LIN {X 0,Y 411.148,Z 377.722,A -85,B 0,C 180,E1 -10646.387,E2 -10646.387} C_VEL
LIN {X 0,Y 411.477,Z 371.571,A -85,B 0,C 180,E1 -10649.691,E2 -10649.691} C_VEL
LIN {X 0,Y 411.355,Z 369.248,A -85,B 0,C 180,E1 -10651.013,E2 -10651.013} C_VEL
LIN {X 0,Y 411.215,Z 369.265,A -85,B 0,C 180,E1 -10654.879,E2 -10654.879} C_VEL
LIN {X 0,Y 411.214,Z 369.262,A -85,B 0,C 180,E1 -10658.17,E2 -10658.17} C_VEL
LIN {X 0,Y 411.167,Z 369.269,A -85,B 0,C 180,E1 -10661.228,E2 -10661.228} C_VEL
LIN {X 0,Y 411.18,Z 369.267,A -85,B 0,C 180,E1 -10664.49,E2 -10664.49} C_VEL
LIN {X 0,Y 411.182,Z 369.267,A -85,B 0,C 180,E1 -10668.195,E2 -10668.195} C_VEL
LIN {X 0,Y 411.22,Z 369.263,A -85,B 0,C 180,E1 -10670.776,E2 -10670.776} C_VEL
LIN {X 0,Y 411.201,Z 369.266,A -85,B 0,C 180,E1 -10674.471,E2 -10674.471} C_VEL
LIN {X 0,Y 411.21,Z 369.263,A -85,B 0,C 180,E1 -10676.873,E2 -10676.873} C_VEL
LIN {X 0,Y 411.236,Z 369.261,A -85,B 0,C 180,E1 -10680.644,E2 -10680.644} C_VEL
LIN {X 0,Y 411.24,Z 369.258,A -85,B 0,C 180,E1 -10683.619,E2 -10683.619} C_VEL
LIN {X 0,Y 411.206,Z 369.263,A -85,B 0,C 180,E1 -10686.852,E2 -10686.852} C_VEL
LIN {X 0,Y 411.219,Z 369.264,A -85,B 0,C 180,E1 -10690.05,E2 -10690.05} C_VEL
LIN {X 0,Y 411.267,Z 369.255,A -85,B 0,C 180,E1 -10693.131,E2 -10693.131} C_VEL
LIN {X 0,Y 411.309,Z 369.248,A -85,B 0,C 180,E1 -10696.896,E2 -10696.896} C_VEL
LIN {X 0,Y 411.296,Z 369.254,A -85,B 0,C 180,E1 -10700.161,E2 -10700.161} C_VEL
LIN {X 0,Y 411.456,Z 369.232,A -85,B 0,C 180,E1 -10703.133,E2 -10703.133} C_VEL
LIN {X 0,Y 411.313,Z 369.249,A -85,B 0,C 180,E1 -10705.099,E2 -10705.099} C_VEL
LIN {X 0,Y 411.515,Z 369.228,A -85,B 0,C 180,E1 -10708.042,E2 -10708.042} C_VEL
LIN {X 0,Y 411.644,Z 369.211,A -85,B 0,C 180,E1 -10710,E2 -10710} C_VEL
LIN {X 0,Y 411.469,Z 369.23,A -85,B 0,C 180,E1 -10712.937,E2 -10712.937} C_VEL
LIN {X 0,Y 411.455,Z 369.231,A -85,B 0,C 180,E1 -10716.867,E2 -10716.867} C_VEL
LIN {X 0,Y 411.308,Z 369.253,A -85,B 0,C 180,E1 -10719.838,E2 -10719.838} C_VEL
LIN {X 0,Y 411.309,Z 369.25,A -85,B 0,C 180,E1 -10723.104,E2 -10723.104} C_VEL
LIN {X 0,Y 411.259,Z 369.255,A -85,B 0,C 180,E1 -10726.756,E2 -10726.756} C_VEL
LIN {X 0,Y 410.624,Z 369.339,A -85,B 0,C 180,E1 -10727.574,E2 -10727.574} C_VEL
LIN {X 0,Y 407.754,Z 369.691,A -85,B 0,C 180,E1 -10728.902,E2 -10728.902} C_VEL
LIN {X 0,Y 405.301,Z 369.999,A -85,B 0,C 180,E1 -10729.974,E2 -10729.974} C_VEL
LIN {X 0,Y 404.247,Z 370.128,A -85,B 0,C 180,E1 -10730.804,E2 -10730.804} C_VEL
LIN {X 0,Y 404.162,Z 370.14,A -85,B 0,C 180,E1 -10731.085,E2 -10731.085} C_VEL
LIN {X 0,Y 404.18,Z 370.138,A -85,B 0,C 180,E1 -10734.665,E2 -10734.665} C_VEL
LIN {X 0,Y 404.198,Z 370.137,A -85,B 0,C 180,E1 -10737.999,E2 -10737.999} C_VEL
LIN {X 0,Y 404.142,Z 370.145,A -85,B 0,C 180,E1 -10741.558,E2 -10741.558} C_VEL
LIN {X 0,Y 404.187,Z 370.139,A -85,B 0,C 180,E1 -10745.016,E2 -10745.016} C_VEL
LIN {X 0,Y 404.16,Z 370.141,A -85,B 0,C 180,E1 -10748.756,E2 -10748.756} C_VEL
LIN {X 0,Y 404.126,Z 370.146,A -85,B 0,C 180,E1 -10751.6,E2 -10751.6} C_VEL
LIN {X 0,Y 404.148,Z 370.142,A -85,B 0,C 180,E1 -10754.522,E2 -10754.522} C_VEL
LIN {X 0,Y 404.139,Z 370.145,A -85,B 0,C 180,E1 -10757.296,E2 -10757.296} C_VEL
LIN {X 0,Y 404.171,Z 370.139,A -85,B 0,C 180,E1 -10759.955,E2 -10759.955} C_VEL
LIN {X 0,Y 404.139,Z 370.147,A -85,B 0,C 180,E1 -10763.125,E2 -10763.125} C_VEL
LIN {X 0,Y 404.147,Z 370.142,A -85,B 0,C 180,E1 -10766.188,E2 -10766.188} C_VEL
LIN {X 0,Y 404.148,Z 370.142,A -85,B 0,C 180,E1 -10769.715,E2 -10769.715} C_VEL
LIN {X 0,Y 404.198,Z 370.138,A -85,B 0,C 180,E1 -10773.123,E2 -10773.123} C_VEL
LIN {X 0,Y 404.18,Z 370.138,A -85,B 0,C 180,E1 -10775.334,E2 -10775.334} C_VEL
LIN {X 0,Y 404.142,Z 370.145,A -85,B 0,C 180,E1 -10778.581,E2 -10778.581} C_VEL
LIN {X 0,Y 404.213,Z 370.133,A -85,B 0,C 180,E1 -10781.762,E2 -10781.762} C_VEL
LIN {X 0,Y 404.21,Z 370.137,A -85,B 0,C 180,E1 -10784.882,E2 -10784.882} C_VEL
LIN {X 0,Y 404.273,Z 370.126,A -85,B 0,C 180,E1 -10787.959,E2 -10787.959} C_VEL
LIN {X 0,Y 404.436,Z 370.107,A -85,B 0,C 180,E1 -10792.1,E2 -10792.1} C_VEL
LIN {X 0,Y 404.426,Z 370.107,A -85,B 0,C 180,E1 -10794.015,E2 -10794.015} C_VEL
LIN {X 0,Y 404.483,Z 370.101,A -85,B 0,C 180,E1 -10798.008,E2 -10798.008} C_VEL
LIN {X 0,Y 404.614,Z 370.085,A -85,B 0,C 180,E1 -10800,E2 -10800} C_VEL
LIN {X 0,Y 404.425,Z 370.108,A -85,B 0,C 180,E1 -10802.988,E2 -10802.988} C_VEL
LIN {X 0,Y 404.414,Z 370.108,A -85,B 0,C 180,E1 -10806.987,E2 -10806.987} C_VEL
LIN {X 0,Y 404.261,Z 370.13,A -85,B 0,C 180,E1 -10810.012,E2 -10810.012} C_VEL
LIN {X 0,Y 404.268,Z 370.127,A -85,B 0,C 180,E1 -10813.211,E2 -10813.211} C_VEL
LIN {X 0,Y 404.218,Z 370.132,A -85,B 0,C 180,E1 -10817.007,E2 -10817.007} C_VEL
LIN {X 0,Y 404.166,Z 370.141,A -85,B 0,C 180,E1 -10820.351,E2 -10820.351} C_VEL
LIN {X 0,Y 404.171,Z 370.14,A -85,B 0,C 180,E1 -10823.574,E2 -10823.574} C_VEL
LIN {X 0,Y 404.185,Z 370.138,A -85,B 0,C 180,E1 -10825.766,E2 -10825.766} C_VEL
LIN {X 0,Y 404.197,Z 370.139,A -85,B 0,C 180,E1 -10828,E2 -10828} C_VEL
LIN {X 0,Y 404.141,Z 370.144,A -85,B 0,C 180,E1 -10831.558,E2 -10831.558} C_VEL
LIN {X 0,Y 404.187,Z 370.137,A -85,B 0,C 180,E1 -10835.016,E2 -10835.016} C_VEL
LIN {X 0,Y 404.161,Z 370.139,A -85,B 0,C 180,E1 -10838.756,E2 -10838.756} C_VEL
LIN {X 0,Y 404.143,Z 370.145,A -85,B 0,C 180,E1 -10841.603,E2 -10841.603} C_VEL
LIN {X 0,Y 404.152,Z 370.142,A -85,B 0,C 180,E1 -10844.523,E2 -10844.523} C_VEL
LIN {X 0,Y 404.141,Z 370.144,A -85,B 0,C 180,E1 -10847.296,E2 -10847.296} C_VEL
LIN {X 0,Y 404.17,Z 370.14,A -85,B 0,C 180,E1 -10849.955,E2 -10849.955} C_VEL
LIN {X 0,Y 404.18,Z 370.14,A -85,B 0,C 180,E1 -10853.758,E2 -10853.758} C_VEL
LIN {X 0,Y 404.188,Z 370.32,A -85,B 0,C 180,E1 -10854.162,E2 -10854.162} C_VEL
LIN {X 0,Y 406.436,Z 380.828,A -85,B 0,C 180,E1 -10857.291,E2 -10857.291} C_VEL
LIN {X 0,Y 408.438,Z 390.536,A -85,B 0,C 180,E1 -10860.066,E2 -10860.066} C_VEL
LIN {X 0,Y 408.583,Z 393.722,A -85,B 0,C 180,E1 -10860.927,E2 -10860.927} C_VEL
LIN {X 0,Y 407.037,Z 407.44,A -85,B 0,C 180,E1 -10864.427,E2 -10864.427} C_VEL
LIN {X 0,Y 405.68,Z 422.214,A -85,B 0,C 180,E1 -10868.132,E2 -10868.132} C_VEL
LIN {X 0,Y 404.511,Z 439.114,A -85,B 0,C 180,E1 -10872.299,E2 -10872.299} C_VEL
LIN {X 0,Y 404.238,Z 443.217,A -85,B 0,C 180,E1 -10873.301,E2 -10873.301} C_VEL
LIN {X 0,Y 405.63,Z 458.581,A -85,B 0,C 180,E1 -10873.82,E2 -10873.82} C_VEL
LIN {X 0,Y 406.354,Z 470.143,A -85,B 0,C 180,E1 -10874.386,E2 -10874.386} C_VEL
LIN {X 0,Y 405.709,Z 482.837,A -85,B 0,C 180,E1 -10875.196,E2 -10875.196} C_VEL
LIN {X 0,Y 405.185,Z 494.035,A -85,B 0,C 180,E1 -10876.131,E2 -10876.131} C_VEL
LIN {X 0,Y 404.711,Z 503.184,A -85,B 0,C 180,E1 -10877.081,E2 -10877.081} C_VEL
LIN {X 0,Y 404.142,Z 512.126,A -85,B 0,C 180,E1 -10878.21,E2 -10878.21} C_VEL
LIN {X 0,Y 403.682,Z 520.303,A -85,B 0,C 180,E1 -10879.467,E2 -10879.467} C_VEL
LIN {X 0,Y 403.357,Z 528.26,A -85,B 0,C 180,E1 -10880.978,E2 -10880.978} C_VEL
LIN {X 0,Y 403.201,Z 534.531,A -85,B 0,C 180,E1 -10882.488,E2 -10882.488} C_VEL
LIN {X 0,Y 403.139,Z 539.444,A -85,B 0,C 180,E1 -10883.996,E2 -10883.996} C_VEL
LIN {X 0,Y 403.099,Z 543.144,A -85,B 0,C 180,E1 -10885.5,E2 -10885.5} C_VEL
LIN {X 0,Y 403.268,Z 545.764,A -85,B 0,C 180,E1 -10887.003,E2 -10887.003} C_VEL
LIN {X 0,Y 403.223,Z 546.939,A -85,B 0,C 180,E1 -10888.002,E2 -10888.002} C_VEL
LIN {X 0,Y 403.121,Z 547.631,A -85,B 0,C 180,E1 -10889.001,E2 -10889.001} C_VEL
LIN {X 0,Y 403.102,Z 547.906,A -85,B 0,C 180,E1 -10890,E2 -10890} C_VEL
LIN {X 0,Y 403.123,Z 547.774,A -85,B 0,C 180,E1 -10890.999,E2 -10890.999} C_VEL
LIN {X 0,Y 403.218,Z 547.196,A -85,B 0,C 180,E1 -10891.998,E2 -10891.998} C_VEL
LIN {X 0,Y 403.204,Z 546.167,A -85,B 0,C 180,E1 -10892.998,E2 -10892.998} C_VEL
LIN {X 0,Y 403.116,Z 544.713,A -85,B 0,C 180,E1 -10893.999,E2 -10893.999} C_VEL
LIN {X 0,Y 403.111,Z 541.666,A -85,B 0,C 180,E1 -10895.503,E2 -10895.503} C_VEL
LIN {X 0,Y 403.183,Z 537.532,A -85,B 0,C 180,E1 -10897.009,E2 -10897.009} C_VEL
LIN {X 0,Y 403.332,Z 531.141,A -85,B 0,C 180,E1 -10898.77,E2 -10898.77} C_VEL
LIN {X 0,Y 403.59,Z 524.167,A -85,B 0,C 180,E1 -10900.282,E2 -10900.282} C_VEL
LIN {X 0,Y 404.107,Z 517.08,A -85,B 0,C 180,E1 -10901.537,E2 -10901.537} C_VEL
LIN {X 0,Y 404.66,Z 508.52,A -85,B 0,C 180,E1 -10902.794,E2 -10902.794} C_VEL
LIN {X 0,Y 405.427,Z 497.96,A -85,B 0,C 180,E1 -10904.045,E2 -10904.045} C_VEL
LIN {X 0,Y 406.179,Z 487.574,A -85,B 0,C 180,E1 -10905.043,E2 -10905.043} C_VEL
LIN {X 0,Y 406.997,Z 476.089,A -85,B 0,C 180,E1 -10905.91,E2 -10905.91} C_VEL
LIN {X 0,Y 407.201,Z 467.052,A -85,B 0,C 180,E1 -10906.469,E2 -10906.469} C_VEL
LIN {X 0,Y 406.365,Z 453.454,A -85,B 0,C 180,E1 -10907.152,E2 -10907.152} C_VEL
LIN {X 0,Y 404.671,Z 441.819,A -85,B 0,C 180,E1 -10907.628,E2 -10907.628} C_VEL
LIN {X 0,Y 405.657,Z 428.844,A -85,B 0,C 180,E1 -10910.914,E2 -10910.914} C_VEL
LIN {X 0,Y 406.916,Z 417.346,A -85,B 0,C 180,E1 -10914,E2 -10914} C_VEL
LIN {X 0,Y 408.565,Z 406.517,A -85,B 0,C 180,E1 -10917.119,E2 -10917.119} C_VEL
LIN {X 0,Y 409.97,Z 399.423,A -85,B 0,C 180,E1 -10919.308,E2 -10919.308} C_VEL
LIN {X 0,Y 410.147,Z 396.422,A -85,B 0,C 180,E1 -10920.364,E2 -10920.364} C_VEL
LIN {X 0,Y 408.861,Z 389.269,A -85,B 0,C 180,E1 -10923.371,E2 -10923.371} C_VEL
LIN {X 0,Y 407.709,Z 384.465,A -85,B 0,C 180,E1 -10925.887,E2 -10925.887} C_VEL
LIN {X 0,Y 406.605,Z 379.983,A -85,B 0,C 180,E1 -10928.94,E2 -10928.94} C_VEL
LIN {X 0,Y 406.056,Z 377.657,A -85,B 0,C 180,E1 -10931.125,E2 -10931.125} C_VEL
LIN {X 0,Y 405.542,Z 375.828,A -85,B 0,C 180,E1 -10933.884,E2 -10933.884} C_VEL
LIN {X 0,Y 405.371,Z 375.113,A -85,B 0,C 180,E1 -10936.733,E2 -10936.733} C_VEL
LIN {X 0,Y 405.424,Z 375.549,A -85,B 0,C 180,E1 -10939.707,E2 -10939.707} C_VEL
LIN {X 0,Y 405.674,Z 377.131,A -85,B 0,C 180,E1 -10942.837,E2 -10942.837} C_VEL
LIN {X 0,Y 406.006,Z 378.918,A -85,B 0,C 180,E1 -10945.164,E2 -10945.164} C_VEL
LIN {X 0,Y 406.357,Z 381.647,A -85,B 0,C 180,E1 -10947.937,E2 -10947.937} C_VEL
LIN {X 0,Y 406.342,Z 383.966,A -85,B 0,C 180,E1 -10949.896,E2 -10949.896} C_VEL
LIN {X 0,Y 405.779,Z 388.489,A -85,B 0,C 180,E1 -10953.236,E2 -10953.236} C_VEL
LIN {X 0,Y 405.249,Z 393.854,A -85,B 0,C 180,E1 -10956.803,E2 -10956.803} C_VEL
LIN {X 0,Y 404.742,Z 400.152,A -85,B 0,C 180,E1 -10960.736,E2 -10960.736} C_VEL
LIN {X 0,Y 404.373,Z 405.404,A -85,B 0,C 180,E1 -10963.854,E2 -10963.854} C_VEL
LIN {X 0,Y 404.048,Z 412.145,A -85,B 0,C 180,E1 -10967.697,E2 -10967.697} C_VEL
LIN {X 0,Y 404.018,Z 412.616,A -85,B 0,C 180,E1 -10967.951,E2 -10967.951} C_VEL
LIN {X 0,Y 406.519,Z 423.605,A -85,B 0,C 180,E1 -10968.785,E2 -10968.785} C_VEL
LIN {X 0,Y 407.207,Z 428.2,A -85,B 0,C 180,E1 -10969.182,E2 -10969.182} C_VEL
LIN {X 0,Y 406.611,Z 437.638,A -85,B 0,C 180,E1 -10970.047,E2 -10970.047} C_VEL
LIN {X 0,Y 405.969,Z 446.024,A -85,B 0,C 180,E1 -10971.037,E2 -10971.037} C_VEL
LIN {X 0,Y 405.274,Z 454.119,A -85,B 0,C 180,E1 -10972.276,E2 -10972.276} C_VEL
LIN {X 0,Y 404.79,Z 460.311,A -85,B 0,C 180,E1 -10973.52,E2 -10973.52} C_VEL
LIN {X 0,Y 404.377,Z 464.194,A -85,B 0,C 180,E1 -10974.515,E2 -10974.515} C_VEL
LIN {X 0,Y 404.143,Z 467.219,A -85,B 0,C 180,E1 -10975.512,E2 -10975.512} C_VEL
LIN {X 0,Y 403.552,Z 470.386,A -85,B 0,C 180,E1 -10977.005,E2 -10977.005} C_VEL
LIN {X 0,Y 403.365,Z 471.602,A -85,B 0,C 180,E1 -10978.003,E2 -10978.003} C_VEL
LIN {X 0,Y 403.255,Z 472.146,A -85,B 0,C 180,E1 -10979.001,E2 -10979.001} C_VEL
LIN {X 0,Y 403.193,Z 472.025,A -85,B 0,C 180,E1 -10980,E2 -10980} C_VEL
LIN {X 0,Y 403.192,Z 471.236,A -85,B 0,C 180,E1 -10980.999,E2 -10980.999} C_VEL
LIN {X 0,Y 403.346,Z 468.774,A -85,B 0,C 180,E1 -10982.497,E2 -10982.497} C_VEL
LIN {X 0,Y 403.608,Z 466.231,A -85,B 0,C 180,E1 -10983.494,E2 -10983.494} C_VEL
LIN {X 0,Y 403.853,Z 460.925,A -85,B 0,C 180,E1 -10984.992,E2 -10984.992} C_VEL
LIN {X 0,Y 404.041,Z 454.874,A -85,B 0,C 180,E1 -10986.241,E2 -10986.241} C_VEL
LIN {X 0,Y 404.249,Z 447.598,A -85,B 0,C 180,E1 -10987.399,E2 -10987.399} C_VEL
LIN {X 0,Y 404.594,Z 438.691,A -85,B 0,C 180,E1 -10988.491,E2 -10988.491} C_VEL
LIN {X 0,Y 404.977,Z 429.418,A -85,B 0,C 180,E1 -10989.363,E2 -10989.363} C_VEL
LIN {X 0,Y 405.109,Z 422.751,A -85,B 0,C 180,E1 -10989.864,E2 -10989.864} C_VEL
LIN {X 0,Y 403.584,Z 411.764,A -85,B 0,C 180,E1 -10990.536,E2 -10990.536} C_VEL
LIN {X 0,Y 403.201,Z 408.969,A -85,B 0,C 180,E1 -10990.673,E2 -10990.673} C_VEL
LIN {X 0,Y 403.341,Z 403.119,A -85,B 0,C 180,E1 -10993.605,E2 -10993.605} C_VEL
LIN {X 0,Y 403.527,Z 397.076,A -85,B 0,C 180,E1 -10996.683,E2 -10996.683} C_VEL
LIN {X 0,Y 403.733,Z 389.969,A -85,B 0,C 180,E1 -11000.374,E2 -11000.374} C_VEL
LIN {X 0,Y 403.888,Z 383.868,A -85,B 0,C 180,E1 -11003.592,E2 -11003.592} C_VEL
LIN {X 0,Y 404.111,Z 377.71,A -85,B 0,C 180,E1 -11006.883,E2 -11006.883} C_VEL
LIN {X 0,Y 404.505,Z 371.515,A -85,B 0,C 180,E1 -11010.256,E2 -11010.256} C_VEL
LIN {X 0,Y 404.318,Z 370.125,A -85,B 0,C 180,E1 -11011.14,E2 -11011.14} C_VEL
LIN {X 0,Y 404.185,Z 370.138,A -85,B 0,C 180,E1 -11015.19,E2 -11015.19} C_VEL
LIN {X 0,Y 404.161,Z 370.142,A -85,B 0,C 180,E1 -11018.756,E2 -11018.756} C_VEL
LIN {X 0,Y 404.126,Z 370.144,A -85,B 0,C 180,E1 -11021.6,E2 -11021.6} C_VEL
LIN {X 0,Y 404.15,Z 370.144,A -85,B 0,C 180,E1 -11024.522,E2 -11024.522} C_VEL
LIN {X 0,Y 404.143,Z 370.143,A -85,B 0,C 180,E1 -11027.296,E2 -11027.296} C_VEL
LIN {X 0,Y 404.172,Z 370.139,A -85,B 0,C 180,E1 -11029.955,E2 -11029.955} C_VEL
LIN {X 0,Y 404.139,Z 370.143,A -85,B 0,C 180,E1 -11033.125,E2 -11033.125} C_VEL
LIN {X 0,Y 404.148,Z 370.143,A -85,B 0,C 180,E1 -11036.188,E2 -11036.188} C_VEL
LIN {X 0,Y 404.149,Z 370.142,A -85,B 0,C 180,E1 -11039.715,E2 -11039.715} C_VEL
LIN {X 0,Y 404.198,Z 370.135,A -85,B 0,C 180,E1 -11043.123,E2 -11043.123} C_VEL
LIN {X 0,Y 404.18,Z 370.136,A -85,B 0,C 180,E1 -11045.334,E2 -11045.334} C_VEL
LIN {X 0,Y 404.142,Z 370.144,A -85,B 0,C 180,E1 -11048.581,E2 -11048.581} C_VEL
LIN {X 0,Y 404.214,Z 370.135,A -85,B 0,C 180,E1 -11051.762,E2 -11051.762} C_VEL
LIN {X 0,Y 404.21,Z 370.134,A -85,B 0,C 180,E1 -11054.882,E2 -11054.882} C_VEL
LIN {X 0,Y 404.26,Z 370.13,A -85,B 0,C 180,E1 -11057.958,E2 -11057.958} C_VEL
LIN {X 0,Y 404.408,Z 370.111,A -85,B 0,C 180,E1 -11062.129,E2 -11062.129} C_VEL
LIN {X 0,Y 404.423,Z 370.109,A -85,B 0,C 180,E1 -11064.015,E2 -11064.015} C_VEL
LIN {X 0,Y 404.484,Z 370.104,A -85,B 0,C 180,E1 -11068.008,E2 -11068.008} C_VEL
LIN {X 0,Y 404.613,Z 370.087,A -85,B 0,C 180,E1 -11070,E2 -11070} C_VEL
LIN {X 0,Y 404.426,Z 370.107,A -85,B 0,C 180,E1 -11072.988,E2 -11072.988} C_VEL
LIN {X 0,Y 404.403,Z 370.109,A -85,B 0,C 180,E1 -11076.987,E2 -11076.987} C_VEL
LIN {X 0,Y 404.27,Z 370.128,A -85,B 0,C 180,E1 -11080.011,E2 -11080.011} C_VEL
LIN {X 0,Y 404.27,Z 370.128,A -85,B 0,C 180,E1 -11083.211,E2 -11083.211} C_VEL
LIN {X 0,Y 404.219,Z 370.133,A -85,B 0,C 180,E1 -11087.007,E2 -11087.007} C_VEL
LIN {X 0,Y 404.201,Z 370.134,A -85,B 0,C 180,E1 -11090.35,E2 -11090.35} C_VEL
LIN {X 0,Y 404.162,Z 370.14,A -85,B 0,C 180,E1 -11091.085,E2 -11091.085} C_VEL
LIN {X 0,Y 403.499,Z 370.226,A -85,B 0,C 180,E1 -11091.917,E2 -11091.917} C_VEL
LIN {X 0,Y 400.656,Z 370.581,A -85,B 0,C 180,E1 -11093.27,E2 -11093.27} C_VEL
LIN {X 0,Y 398.255,Z 370.877,A -85,B 0,C 180,E1 -11094.362,E2 -11094.362} C_VEL
LIN {X 0,Y 397.234,Z 371.006,A -85,B 0,C 180,E1 -11095.207,E2 -11095.207} C_VEL
LIN {X 0,Y 397.156,Z 371.015,A -85,B 0,C 180,E1 -11095.493,E2 -11095.493} C_VEL
LIN {X 0,Y 397.125,Z 371.016,A -85,B 0,C 180,E1 -11098.543,E2 -11098.543} C_VEL
LIN {X 0,Y 397.081,Z 371.022,A -85,B 0,C 180,E1 -11102.071,E2 -11102.071} C_VEL
LIN {X 0,Y 397.122,Z 371.019,A -85,B 0,C 180,E1 -11105.503,E2 -11105.503} C_VEL
LIN {X 0,Y 397.134,Z 371.016,A -85,B 0,C 180,E1 -11108.862,E2 -11108.862} C_VEL
LIN {X 0,Y 397.071,Z 371.021,A -85,B 0,C 180,E1 -11112.267,E2 -11112.267} C_VEL
LIN {X 0,Y 397.09,Z 371.024,A -85,B 0,C 180,E1 -11115.069,E2 -11115.069} C_VEL
LIN {X 0,Y 397.068,Z 371.024,A -85,B 0,C 180,E1 -11118.021,E2 -11118.021} C_VEL
LIN {X 0,Y 397.132,Z 371.019,A -85,B 0,C 180,E1 -11121.139,E2 -11121.139} C_VEL
LIN {X 0,Y 397.121,Z 371.017,A -85,B 0,C 180,E1 -11124.497,E2 -11124.497} C_VEL
LIN {X 0,Y 397.08,Z 371.022,A -85,B 0,C 180,E1 -11127.928,E2 -11127.928} C_VEL
LIN {X 0,Y 397.124,Z 371.017,A -85,B 0,C 180,E1 -11131.456,E2 -11131.456} C_VEL
LIN {X 0,Y 397.155,Z 371.013,A -85,B 0,C 180,E1 -11134.487,E2 -11134.487} C_VEL
LIN {X 0,Y 397.112,Z 371.02,A -85,B 0,C 180,E1 -11137.086,E2 -11137.086} C_VEL
LIN {X 0,Y 397.151,Z 371.015,A -85,B 0,C 180,E1 -11140.353,E2 -11140.353} C_VEL
LIN {X 0,Y 397.169,Z 371.01,A -85,B 0,C 180,E1 -11143.553,E2 -11143.553} C_VEL
LIN {X 0,Y 397.231,Z 371.007,A -85,B 0,C 180,E1 -11146.703,E2 -11146.703} C_VEL
LIN {X 0,Y 397.231,Z 371.003,A -85,B 0,C 180,E1 -11149.809,E2 -11149.809} C_VEL
LIN {X 0,Y 397.367,Z 370.989,A -85,B 0,C 180,E1 -11152.888,E2 -11152.888} C_VEL
LIN {X 0,Y 397.256,Z 371.001,A -85,B 0,C 180,E1 -11154.925,E2 -11154.925} C_VEL
LIN {X 0,Y 397.452,Z 370.976,A -85,B 0,C 180,E1 -11157.973,E2 -11157.973} C_VEL
LIN {X 0,Y 397.584,Z 370.961,A -85,B 0,C 180,E1 -11160,E2 -11160} C_VEL
LIN {X 0,Y 397.384,Z 370.985,A -85,B 0,C 180,E1 -11163.041,E2 -11163.041} C_VEL
LIN {X 0,Y 397.366,Z 370.985,A -85,B 0,C 180,E1 -11167.112,E2 -11167.112} C_VEL
LIN {X 0,Y 397.22,Z 371.008,A -85,B 0,C 180,E1 -11170.191,E2 -11170.191} C_VEL
LIN {X 0,Y 397.228,Z 371.003,A -85,B 0,C 180,E1 -11173.321,E2 -11173.321} C_VEL
LIN {X 0,Y 397.184,Z 371.007,A -85,B 0,C 180,E1 -11177.155,E2 -11177.155} C_VEL
LIN {X 0,Y 397.105,Z 371.02,A -85,B 0,C 180,E1 -11180.73,E2 -11180.73} C_VEL
LIN {X 0,Y 397.135,Z 371.017,A -85,B 0,C 180,E1 -11184.018,E2 -11184.018} C_VEL
LIN {X 0,Y 397.196,Z 371.007,A -85,B 0,C 180,E1 -11187.39,E2 -11187.39} C_VEL
LIN {X 0,Y 397.08,Z 371.021,A -85,B 0,C 180,E1 -11190.882,E2 -11190.882} C_VEL
LIN {X 0,Y 397.128,Z 371.017,A -85,B 0,C 180,E1 -11194.493,E2 -11194.493} C_VEL
LIN {X 0,Y 397.109,Z 371.019,A -85,B 0,C 180,E1 -11198.274,E2 -11198.274} C_VEL
LIN {X 0,Y 397.108,Z 371.017,A -85,B 0,C 180,E1 -11200.906,E2 -11200.906} C_VEL
LIN {X 0,Y 397.106,Z 371.022,A -85,B 0,C 180,E1 -11203.648,E2 -11203.648} C_VEL
LIN {X 0,Y 397.107,Z 371.019,A -85,B 0,C 180,E1 -11206.521,E2 -11206.521} C_VEL
LIN {X 0,Y 397.114,Z 371.015,A -85,B 0,C 180,E1 -11210.423,E2 -11210.423} C_VEL
LIN {X 0,Y 397.152,Z 371.109,A -85,B 0,C 180,E1 -11213.8,E2 -11213.8} C_VEL
LIN {X 0,Y 399.3,Z 381.365,A -85,B 0,C 180,E1 -11216.933,E2 -11216.933} C_VEL
LIN {X 0,Y 401.539,Z 392.137,A -85,B 0,C 180,E1 -11220.078,E2 -11220.078} C_VEL
LIN {X 0,Y 401.478,Z 395.829,A -85,B 0,C 180,E1 -11221.077,E2 -11221.077} C_VEL
LIN {X 0,Y 399.967,Z 408.977,A -85,B 0,C 180,E1 -11224.501,E2 -11224.501} C_VEL
LIN {X 0,Y 398.567,Z 423.688,A -85,B 0,C 180,E1 -11228.266,E2 -11228.266} C_VEL
LIN {X 0,Y 397.458,Z 439.439,A -85,B 0,C 180,E1 -11232.241,E2 -11232.241} C_VEL
LIN {X 0,Y 397.176,Z 442.964,A -85,B 0,C 180,E1 -11233.121,E2 -11233.121} C_VEL
LIN {X 0,Y 398.535,Z 458.171,A -85,B 0,C 180,E1 -11233.644,E2 -11233.644} C_VEL
LIN {X 0,Y 399.349,Z 469.923,A -85,B 0,C 180,E1 -11234.236,E2 -11234.236} C_VEL
LIN {X 0,Y 398.687,Z 482.543,A -85,B 0,C 180,E1 -11235.06,E2 -11235.06} C_VEL
LIN {X 0,Y 398.166,Z 492.99,A -85,B 0,C 180,E1 -11235.943,E2 -11235.943} C_VEL
LIN {X 0,Y 397.653,Z 502.792,A -85,B 0,C 180,E1 -11236.977,E2 -11236.977} C_VEL
LIN {X 0,Y 397.038,Z 512.6,A -85,B 0,C 180,E1 -11238.255,E2 -11238.255} C_VEL
LIN {X 0,Y 396.558,Z 520.596,A -85,B 0,C 180,E1 -11239.534,E2 -11239.534} C_VEL
LIN {X 0,Y 396.285,Z 528.335,A -85,B 0,C 180,E1 -11241.073,E2 -11241.073} C_VEL
LIN {X 0,Y 396.145,Z 533.555,A -85,B 0,C 180,E1 -11242.354,E2 -11242.354} C_VEL
LIN {X 0,Y 396.077,Z 538.537,A -85,B 0,C 180,E1 -11243.889,E2 -11243.889} C_VEL
LIN {X 0,Y 396.026,Z 542.296,A -85,B 0,C 180,E1 -11245.42,E2 -11245.42} C_VEL
LIN {X 0,Y 396.193,Z 544.968,A -85,B 0,C 180,E1 -11246.95,E2 -11246.95} C_VEL
LIN {X 0,Y 396.175,Z 546.171,A -85,B 0,C 180,E1 -11247.967,E2 -11247.967} C_VEL
LIN {X 0,Y 396.069,Z 546.905,A -85,B 0,C 180,E1 -11248.983,E2 -11248.983} C_VEL
LIN {X 0,Y 396.047,Z 547.197,A -85,B 0,C 180,E1 -11250,E2 -11250} C_VEL
LIN {X 0,Y 396.071,Z 547.084,A -85,B 0,C 180,E1 -11251.017,E2 -11251.017} C_VEL
LIN {X 0,Y 396.168,Z 546.544,A -85,B 0,C 180,E1 -11252.033,E2 -11252.033} C_VEL
LIN {X 0,Y 396.133,Z 545.529,A -85,B 0,C 180,E1 -11253.051,E2 -11253.051} C_VEL
LIN {X 0,Y 396.026,Z 544.09,A -85,B 0,C 180,E1 -11254.071,E2 -11254.071} C_VEL
LIN {X 0,Y 396.029,Z 541.078,A -85,B 0,C 180,E1 -11255.601,E2 -11255.601} C_VEL
LIN {X 0,Y 396.094,Z 536.979,A -85,B 0,C 180,E1 -11257.135,E2 -11257.135} C_VEL
LIN {X 0,Y 396.258,Z 530.656,A -85,B 0,C 180,E1 -11258.928,E2 -11258.928} C_VEL
LIN {X 0,Y 396.563,Z 523.736,A -85,B 0,C 180,E1 -11260.466,E2 -11260.466} C_VEL
LIN {X 0,Y 397.191,Z 515.147,A -85,B 0,C 180,E1 -11262,E2 -11262} C_VEL
LIN {X 0,Y 397.959,Z 504.93,A -85,B 0,C 180,E1 -11263.457,E2 -11263.457} C_VEL
LIN {X 0,Y 398.803,Z 494.215,A -85,B 0,C 180,E1 -11264.675,E2 -11264.675} C_VEL
LIN {X 0,Y 399.701,Z 483.079,A -85,B 0,C 180,E1 -11265.685,E2 -11265.685} C_VEL
LIN {X 0,Y 400.516,Z 470.981,A -85,B 0,C 180,E1 -11266.54,E2 -11266.54} C_VEL
LIN {X 0,Y 399.96,Z 457.525,A -85,B 0,C 180,E1 -11267.307,E2 -11267.307} C_VEL
LIN {X 0,Y 398.341,Z 445.046,A -85,B 0,C 180,E1 -11267.866,E2 -11267.866} C_VEL
LIN {X 0,Y 397.719,Z 441.419,A -85,B 0,C 180,E1 -11268.03,E2 -11268.03} C_VEL
LIN {X 0,Y 398.761,Z 429.221,A -85,B 0,C 180,E1 -11271.217,E2 -11271.217} C_VEL
LIN {X 0,Y 400.134,Z 417.815,A -85,B 0,C 180,E1 -11274.378,E2 -11274.378} C_VEL
LIN {X 0,Y 401.942,Z 406.996,A -85,B 0,C 180,E1 -11277.604,E2 -11277.604} C_VEL
LIN {X 0,Y 403.332,Z 400.284,A -85,B 0,C 180,E1 -11279.775,E2 -11279.775} C_VEL
LIN {X 0,Y 403.231,Z 397.501,A -85,B 0,C 180,E1 -11280.818,E2 -11280.818} C_VEL
LIN {X 0,Y 402.173,Z 391.559,A -85,B 0,C 180,E1 -11283.421,E2 -11283.421} C_VEL
LIN {X 0,Y 401.356,Z 387.958,A -85,B 0,C 180,E1 -11285.3,E2 -11285.3} C_VEL
LIN {X 0,Y 400.284,Z 383.865,A -85,B 0,C 180,E1 -11287.917,E2 -11287.917} C_VEL
LIN {X 0,Y 399.524,Z 380.487,A -85,B 0,C 180,E1 -11290.851,E2 -11290.851} C_VEL
LIN {X 0,Y 398.956,Z 378.458,A -85,B 0,C 180,E1 -11293.759,E2 -11293.759} C_VEL
LIN {X 0,Y 398.742,Z 377.643,A -85,B 0,C 180,E1 -11296.576,E2 -11296.576} C_VEL
LIN {X 0,Y 398.734,Z 377.844,A -85,B 0,C 180,E1 -11299.296,E2 -11299.296} C_VEL
LIN {X 0,Y 398.918,Z 379.158,A -85,B 0,C 180,E1 -11302.448,E2 -11302.448} C_VEL
LIN {X 0,Y 399.292,Z 381.544,A -85,B 0,C 180,E1 -11305.72,E2 -11305.72} C_VEL
LIN {X 0,Y 399.546,Z 383.865,A -85,B 0,C 180,E1 -11308.15,E2 -11308.15} C_VEL
LIN {X 0,Y 399.387,Z 386.611,A -85,B 0,C 180,E1 -11310.481,E2 -11310.481} C_VEL
LIN {X 0,Y 398.771,Z 391.337,A -85,B 0,C 180,E1 -11314.006,E2 -11314.006} C_VEL
LIN {X 0,Y 398.266,Z 396,A -85,B 0,C 180,E1 -11317.156,E2 -11317.156} C_VEL
LIN {X 0,Y 397.825,Z 401.056,A -85,B 0,C 180,E1 -11320.388,E2 -11320.388} C_VEL
LIN {X 0,Y 397.42,Z 406.276,A -85,B 0,C 180,E1 -11323.564,E2 -11323.564} C_VEL
LIN {X 0,Y 397.069,Z 413.123,A -85,B 0,C 180,E1 -11327.542,E2 -11327.542} C_VEL
LIN {X 0,Y 399.447,Z 423.074,A -85,B 0,C 180,E1 -11328.327,E2 -11328.327} C_VEL
LIN {X 0,Y 400.458,Z 429.057,A -85,B 0,C 180,E1 -11328.869,E2 -11328.869} C_VEL
LIN {X 0,Y 399.796,Z 439.511,A -85,B 0,C 180,E1 -11329.875,E2 -11329.875} C_VEL
LIN {X 0,Y 399.099,Z 447.635,A -85,B 0,C 180,E1 -11330.881,E2 -11330.881} C_VEL
LIN {X 0,Y 398.356,Z 455.522,A -85,B 0,C 180,E1 -11332.141,E2 -11332.141} C_VEL
LIN {X 0,Y 397.844,Z 461.536,A -85,B 0,C 180,E1 -11333.407,E2 -11333.407} C_VEL
LIN {X 0,Y 397.408,Z 465.3,A -85,B 0,C 180,E1 -11334.418,E2 -11334.418} C_VEL
LIN {X 0,Y 397.132,Z 468.225,A -85,B 0,C 180,E1 -11335.432,E2 -11335.432} C_VEL
LIN {X 0,Y 396.519,Z 471.276,A -85,B 0,C 180,E1 -11336.952,E2 -11336.952} C_VEL
LIN {X 0,Y 396.318,Z 472.426,A -85,B 0,C 180,E1 -11337.968,E2 -11337.968} C_VEL
LIN {X 0,Y 396.197,Z 472.903,A -85,B 0,C 180,E1 -11338.984,E2 -11338.984} C_VEL
LIN {X 0,Y 396.133,Z 472.715,A -85,B 0,C 180,E1 -11340,E2 -11340} C_VEL
LIN {X 0,Y 396.136,Z 471.858,A -85,B 0,C 180,E1 -11341.017,E2 -11341.017} C_VEL
LIN {X 0,Y 396.296,Z 469.291,A -85,B 0,C 180,E1 -11342.541,E2 -11342.541} C_VEL
LIN {X 0,Y 396.562,Z 466.677,A -85,B 0,C 180,E1 -11343.556,E2 -11343.556} C_VEL
LIN {X 0,Y 396.798,Z 461.261,A -85,B 0,C 180,E1 -11345.081,E2 -11345.081} C_VEL
LIN {X 0,Y 396.98,Z 455.119,A -85,B 0,C 180,E1 -11346.353,E2 -11346.353} C_VEL
LIN {X 0,Y 397.189,Z 448.293,A -85,B 0,C 180,E1 -11347.454,E2 -11347.454} C_VEL
LIN {X 0,Y 397.521,Z 439.91,A -85,B 0,C 180,E1 -11348.515,E2 -11348.515} C_VEL
LIN {X 0,Y 397.884,Z 430.851,A -85,B 0,C 180,E1 -11349.404,E2 -11349.404} C_VEL
LIN {X 0,Y 397.997,Z 422.554,A -85,B 0,C 180,E1 -11350.043,E2 -11350.043} C_VEL
LIN {X 0,Y 396.389,Z 411.319,A -85,B 0,C 180,E1 -11350.729,E2 -11350.729} C_VEL
LIN {X 0,Y 396.158,Z 409.169,A -85,B 0,C 180,E1 -11350.865,E2 -11350.865} C_VEL
LIN {X 0,Y 396.295,Z 403.284,A -85,B 0,C 180,E1 -11353.852,E2 -11353.852} C_VEL
LIN {X 0,Y 396.47,Z 397.521,A -85,B 0,C 180,E1 -11356.817,E2 -11356.817} C_VEL
LIN {X 0,Y 396.678,Z 391.222,A -85,B 0,C 180,E1 -11360.113,E2 -11360.113} C_VEL
LIN {X 0,Y 396.839,Z 384.897,A -85,B 0,C 180,E1 -11363.483,E2 -11363.483} C_VEL
LIN {X 0,Y 397.086,Z 378.715,A -85,B 0,C 180,E1 -11366.829,E2 -11366.829} C_VEL
LIN {X 0,Y 397.432,Z 373.039,A -85,B 0,C 180,E1 -11369.946,E2 -11369.946} C_VEL
LIN {X 0,Y 397.295,Z 371,A -85,B 0,C 180,E1 -11371.16,E2 -11371.16} C_VEL
LIN {X 0,Y 397.13,Z 371.017,A -85,B 0,C 180,E1 -11374.493,E2 -11374.493} C_VEL
LIN {X 0,Y 397.109,Z 371.019,A -85,B 0,C 180,E1 -11378.275,E2 -11378.275} C_VEL
LIN {X 0,Y 397.092,Z 371.024,A -85,B 0,C 180,E1 -11380.909,E2 -11380.909} C_VEL
LIN {X 0,Y 397.104,Z 371.017,A -85,B 0,C 180,E1 -11383.648,E2 -11383.648} C_VEL
LIN {X 0,Y 397.108,Z 371.022,A -85,B 0,C 180,E1 -11386.521,E2 -11386.521} C_VEL
LIN {X 0,Y 397.117,Z 371.02,A -85,B 0,C 180,E1 -11390.423,E2 -11390.423} C_VEL
LIN {X 0,Y 397.111,Z 371.019,A -85,B 0,C 180,E1 -11394.265,E2 -11394.265} C_VEL
LIN {X 0,Y 397.118,Z 371.019,A -85,B 0,C 180,E1 -11396.727,E2 -11396.727} C_VEL
LIN {X 0,Y 397.128,Z 371.018,A -85,B 0,C 180,E1 -11400.296,E2 -11400.296} C_VEL
LIN {X 0,Y 397.198,Z 371.011,A -85,B 0,C 180,E1 -11402.61,E2 -11402.61} C_VEL
LIN {X 0,Y 397.135,Z 371.015,A -85,B 0,C 180,E1 -11405.982,E2 -11405.982} C_VEL
LIN {X 0,Y 397.142,Z 371.015,A -85,B 0,C 180,E1 -11409.705,E2 -11409.705} C_VEL
LIN {X 0,Y 397.185,Z 371.01,A -85,B 0,C 180,E1 -11412.845,E2 -11412.845} C_VEL
LIN {X 0,Y 397.232,Z 371.003,A -85,B 0,C 180,E1 -11416.703,E2 -11416.703} C_VEL
LIN {X 0,Y 397.221,Z 371.007,A -85,B 0,C 180,E1 -11419.809,E2 -11419.809} C_VEL
LIN {X 0,Y 397.353,Z 370.988,A -85,B 0,C 180,E1 -11422.888,E2 -11422.888} C_VEL
LIN {X 0,Y 397.257,Z 371,A -85,B 0,C 180,E1 -11424.925,E2 -11424.925} C_VEL
LIN {X 0,Y 397.453,Z 370.979,A -85,B 0,C 180,E1 -11427.973,E2 -11427.973} C_VEL
LIN {X 0,Y 397.583,Z 370.962,A -85,B 0,C 180,E1 -11430,E2 -11430} C_VEL
LIN {X 0,Y 397.384,Z 370.984,A -85,B 0,C 180,E1 -11433.041,E2 -11433.041} C_VEL
LIN {X 0,Y 397.374,Z 370.989,A -85,B 0,C 180,E1 -11436.091,E2 -11436.091} C_VEL
LIN {X 0,Y 397.26,Z 370.998,A -85,B 0,C 180,E1 -11439.162,E2 -11439.162} C_VEL
LIN {X 0,Y 397.223,Z 371.006,A -85,B 0,C 180,E1 -11442.258,E2 -11442.258} C_VEL
LIN {X 0,Y 397.183,Z 371.011,A -85,B 0,C 180,E1 -11445.392,E2 -11445.392} C_VEL
LIN {X 0,Y 397.175,Z 371.009,A -85,B 0,C 180,E1 -11448.573,E2 -11448.573} C_VEL
LIN {X 0,Y 397.114,Z 371.02,A -85,B 0,C 180,E1 -11451.818,E2 -11451.818} C_VEL
LIN {X 0,Y 397.156,Z 371.015,A -85,B 0,C 180,E1 -11455.493,E2 -11455.493} C_VEL
LIN {X 0,Y 396.49,Z 371.1,A -85,B 0,C 180,E1 -11456.339,E2 -11456.339} C_VEL
LIN {X 0,Y 393.596,Z 371.46,A -85,B 0,C 180,E1 -11457.714,E2 -11457.714} C_VEL
LIN {X 0,Y 391.151,Z 371.76,A -85,B 0,C 180,E1 -11458.824,E2 -11458.824} C_VEL
LIN {X 0,Y 390.118,Z 371.892,A -85,B 0,C 180,E1 -11459.684,E2 -11459.684} C_VEL
LIN {X 0,Y 390.043,Z 371.897,A -85,B 0,C 180,E1 -11459.975,E2 -11459.975} C_VEL
LIN {X 0,Y 390.046,Z 371.898,A -85,B 0,C 180,E1 -11462.721,E2 -11462.721} C_VEL
LIN {X 0,Y 390.058,Z 371.899,A -85,B 0,C 180,E1 -11465.825,E2 -11465.825} C_VEL
LIN {X 0,Y 390.073,Z 371.897,A -85,B 0,C 180,E1 -11469.218,E2 -11469.218} C_VEL
LIN {X 0,Y 390.045,Z 371.897,A -85,B 0,C 180,E1 -11472.374,E2 -11472.374} C_VEL
LIN {X 0,Y 390.047,Z 371.9,A -85,B 0,C 180,E1 -11475.354,E2 -11475.354} C_VEL
LIN {X 0,Y 390.033,Z 371.899,A -85,B 0,C 180,E1 -11478.187,E2 -11478.187} C_VEL
LIN {X 0,Y 390.092,Z 371.894,A -85,B 0,C 180,E1 -11480.908,E2 -11480.908} C_VEL
LIN {X 0,Y 390.087,Z 371.895,A -85,B 0,C 180,E1 -11484.793,E2 -11484.793} C_VEL
LIN {X 0,Y 390.026,Z 371.902,A -85,B 0,C 180,E1 -11488.496,E2 -11488.496} C_VEL
LIN {X 0,Y 390.119,Z 371.888,A -85,B 0,C 180,E1 -11492.07,E2 -11492.07} C_VEL
LIN {X 0,Y 390.082,Z 371.894,A -85,B 0,C 180,E1 -11495.519,E2 -11495.519} C_VEL
LIN {X 0,Y 390.058,Z 371.899,A -85,B 0,C 180,E1 -11498.878,E2 -11498.878} C_VEL
LIN {X 0,Y 390.13,Z 371.888,A -85,B 0,C 180,E1 -11502.167,E2 -11502.167} C_VEL
LIN {X 0,Y 390.149,Z 371.885,A -85,B 0,C 180,E1 -11505.393,E2 -11505.393} C_VEL
LIN {X 0,Y 390.162,Z 371.887,A -85,B 0,C 180,E1 -11508.571,E2 -11508.571} C_VEL
LIN {X 0,Y 390.346,Z 371.861,A -85,B 0,C 180,E1 -11511.993,E2 -11511.993} C_VEL
LIN {X 0,Y 390.228,Z 371.878,A -85,B 0,C 180,E1 -11514.833,E2 -11514.833} C_VEL
LIN {X 0,Y 390.42,Z 371.852,A -85,B 0,C 180,E1 -11517.937,E2 -11517.937} C_VEL
LIN {X 0,Y 390.553,Z 371.836,A -85,B 0,C 180,E1 -11520,E2 -11520} C_VEL
LIN {X 0,Y 390.318,Z 371.865,A -85,B 0,C 180,E1 -11523.096,E2 -11523.096} C_VEL
LIN {X 0,Y 390.332,Z 371.865,A -85,B 0,C 180,E1 -11526.202,E2 -11526.202} C_VEL
LIN {X 0,Y 390.317,Z 371.869,A -85,B 0,C 180,E1 -11528.282,E2 -11528.282} C_VEL
LIN {X 0,Y 390.173,Z 371.885,A -85,B 0,C 180,E1 -11532.483,E2 -11532.483} C_VEL
LIN {X 0,Y 390.141,Z 371.887,A -85,B 0,C 180,E1 -11535.677,E2 -11535.677} C_VEL
LIN {X 0,Y 390.107,Z 371.89,A -85,B 0,C 180,E1 -11538.922,E2 -11538.922} C_VEL
LIN {X 0,Y 390.042,Z 371.901,A -85,B 0,C 180,E1 -11542.234,E2 -11542.234} C_VEL
LIN {X 0,Y 390.121,Z 371.89,A -85,B 0,C 180,E1 -11545.743,E2 -11545.743} C_VEL
LIN {X 0,Y 390.06,Z 371.895,A -85,B 0,C 180,E1 -11549.109,E2 -11549.109} C_VEL
LIN {X 0,Y 390.044,Z 371.898,A -85,B 0,C 180,E1 -11552.721,E2 -11552.721} C_VEL
LIN {X 0,Y 390.059,Z 371.899,A -85,B 0,C 180,E1 -11555.826,E2 -11555.826} C_VEL
LIN {X 0,Y 390.074,Z 371.894,A -85,B 0,C 180,E1 -11559.219,E2 -11559.219} C_VEL
LIN {X 0,Y 390.052,Z 371.898,A -85,B 0,C 180,E1 -11562.376,E2 -11562.376} C_VEL
LIN {X 0,Y 390.05,Z 371.9,A -85,B 0,C 180,E1 -11565.355,E2 -11565.355} C_VEL
LIN {X 0,Y 390.034,Z 371.901,A -85,B 0,C 180,E1 -11568.187,E2 -11568.187} C_VEL
LIN {X 0,Y 390.089,Z 371.89,A -85,B 0,C 180,E1 -11570.907,E2 -11570.907} C_VEL
LIN {X 0,Y 390.1,Z 372,A -85,B 0,C 180,E1 -11573.481,E2 -11573.481} C_VEL
LIN {X 0,Y 392.363,Z 382.755,A -85,B 0,C 180,E1 -11576.826,E2 -11576.826} C_VEL
LIN {X 0,Y 394.286,Z 391.737,A -85,B 0,C 180,E1 -11579.512,E2 -11579.512} C_VEL
LIN {X 0,Y 394.62,Z 396.174,A -85,B 0,C 180,E1 -11580.77,E2 -11580.77} C_VEL
LIN {X 0,Y 392.998,Z 409.433,A -85,B 0,C 180,E1 -11584.3,E2 -11584.3} C_VEL
LIN {X 0,Y 391.556,Z 424.065,A -85,B 0,C 180,E1 -11588.134,E2 -11588.134} C_VEL
LIN {X 0,Y 390.403,Z 439.717,A -85,B 0,C 180,E1 -11592.18,E2 -11592.18} C_VEL
LIN {X 0,Y 390.146,Z 442.929,A -85,B 0,C 180,E1 -11592.964,E2 -11592.964} C_VEL
LIN {X 0,Y 391.273,Z 456.792,A -85,B 0,C 180,E1 -11593.433,E2 -11593.433} C_VEL
LIN {X 0,Y 392.213,Z 468.352,A -85,B 0,C 180,E1 -11594.008,E2 -11594.008} C_VEL
LIN {X 0,Y 391.918,Z 478.668,A -85,B 0,C 180,E1 -11594.663,E2 -11594.663} C_VEL
LIN {X 0,Y 391.326,Z 489.74,A -85,B 0,C 180,E1 -11595.56,E2 -11595.56} C_VEL
LIN {X 0,Y 390.678,Z 500.059,A -85,B 0,C 180,E1 -11596.608,E2 -11596.608} C_VEL
LIN {X 0,Y 390.05,Z 509.394,A -85,B 0,C 180,E1 -11597.777,E2 -11597.777} C_VEL
LIN {X 0,Y 389.648,Z 517.848,A -85,B 0,C 180,E1 -11599.083,E2 -11599.083} C_VEL
LIN {X 0,Y 389.277,Z 526.036,A -85,B 0,C 180,E1 -11600.649,E2 -11600.649} C_VEL
LIN {X 0,Y 389.073,Z 532.539,A -85,B 0,C 180,E1 -11602.214,E2 -11602.214} C_VEL
LIN {X 0,Y 389.011,Z 537.599,A -85,B 0,C 180,E1 -11603.777,E2 -11603.777} C_VEL
LIN {X 0,Y 388.957,Z 541.424,A -85,B 0,C 180,E1 -11605.336,E2 -11605.336} C_VEL
LIN {X 0,Y 389.12,Z 544.153,A -85,B 0,C 180,E1 -11606.894,E2 -11606.894} C_VEL
LIN {X 0,Y 389.127,Z 545.383,A -85,B 0,C 180,E1 -11607.93,E2 -11607.93} C_VEL
LIN {X 0,Y 389.019,Z 546.166,A -85,B 0,C 180,E1 -11608.965,E2 -11608.965} C_VEL
LIN {X 0,Y 388.994,Z 546.483,A -85,B 0,C 180,E1 -11610,E2 -11610} C_VEL
LIN {X 0,Y 389.021,Z 546.39,A -85,B 0,C 180,E1 -11611.035,E2 -11611.035} C_VEL
LIN {X 0,Y 389.118,Z 545.886,A -85,B 0,C 180,E1 -11612.07,E2 -11612.07} C_VEL
LIN {X 0,Y 389.062,Z 544.894,A -85,B 0,C 180,E1 -11613.107,E2 -11613.107} C_VEL
LIN {X 0,Y 388.937,Z 543.474,A -85,B 0,C 180,E1 -11614.145,E2 -11614.145} C_VEL
LIN {X 0,Y 388.928,Z 540.503,A -85,B 0,C 180,E1 -11615.704,E2 -11615.704} C_VEL
LIN {X 0,Y 389.015,Z 536.447,A -85,B 0,C 180,E1 -11617.265,E2 -11617.265} C_VEL
LIN {X 0,Y 389.187,Z 530.201,A -85,B 0,C 180,E1 -11619.091,E2 -11619.091} C_VEL
LIN {X 0,Y 389.554,Z 523.352,A -85,B 0,C 180,E1 -11620.657,E2 -11620.657} C_VEL
LIN {X 0,Y 390.213,Z 514.864,A -85,B 0,C 180,E1 -11622.218,E2 -11622.218} C_VEL
LIN {X 0,Y 390.914,Z 506.137,A -85,B 0,C 180,E1 -11623.516,E2 -11623.516} C_VEL
LIN {X 0,Y 391.814,Z 495.447,A -85,B 0,C 180,E1 -11624.809,E2 -11624.809} C_VEL
LIN {X 0,Y 392.753,Z 484.797,A -85,B 0,C 180,E1 -11625.836,E2 -11625.836} C_VEL
LIN {X 0,Y 393.658,Z 473.304,A -85,B 0,C 180,E1 -11626.713,E2 -11626.713} C_VEL
LIN {X 0,Y 393.356,Z 461.227,A -85,B 0,C 180,E1 -11627.474,E2 -11627.474} C_VEL
LIN {X 0,Y 392.396,Z 450.462,A -85,B 0,C 180,E1 -11628.024,E2 -11628.024} C_VEL
LIN {X 0,Y 390.811,Z 441.051,A -85,B 0,C 180,E1 -11628.459,E2 -11628.459} C_VEL
LIN {X 0,Y 392.191,Z 427.545,A -85,B 0,C 180,E1 -11632.106,E2 -11632.106} C_VEL
LIN {X 0,Y 393.989,Z 414.502,A -85,B 0,C 180,E1 -11635.915,E2 -11635.915} C_VEL
LIN {X 0,Y 396.112,Z 404.27,A -85,B 0,C 180,E1 -11639.173,E2 -11639.173} C_VEL
LIN {X 0,Y 396.577,Z 400.969,A -85,B 0,C 180,E1 -11640.336,E2 -11640.336} C_VEL
LIN {X 0,Y 395.714,Z 395.296,A -85,B 0,C 180,E1 -11642.768,E2 -11642.768} C_VEL
LIN {X 0,Y 394.813,Z 390.9,A -85,B 0,C 180,E1 -11645.031,E2 -11645.031} C_VEL
LIN {X 0,Y 393.572,Z 386.033,A -85,B 0,C 180,E1 -11648.214,E2 -11648.214} C_VEL
LIN {X 0,Y 393.079,Z 383.835,A -85,B 0,C 180,E1 -11650.065,E2 -11650.065} C_VEL
LIN {X 0,Y 392.461,Z 381.524,A -85,B 0,C 180,E1 -11652.882,E2 -11652.882} C_VEL
LIN {X 0,Y 392.132,Z 380.291,A -85,B 0,C 180,E1 -11655.8,E2 -11655.8} C_VEL
LIN {X 0,Y 392.047,Z 380.189,A -85,B 0,C 180,E1 -11658.843,E2 -11658.843} C_VEL
LIN {X 0,Y 392.188,Z 381.247,A -85,B 0,C 180,E1 -11662.044,E2 -11662.044} C_VEL
LIN {X 0,Y 392.489,Z 383.451,A -85,B 0,C 180,E1 -11665.456,E2 -11665.456} C_VEL
LIN {X 0,Y 392.728,Z 385.283,A -85,B 0,C 180,E1 -11667.53,E2 -11667.53} C_VEL
LIN {X 0,Y 392.627,Z 387.874,A -85,B 0,C 180,E1 -11669.921,E2 -11669.921} C_VEL
LIN {X 0,Y 392.184,Z 390.746,A -85,B 0,C 180,E1 -11672.23,E2 -11672.23} C_VEL
LIN {X 0,Y 391.567,Z 395.392,A -85,B 0,C 180,E1 -11675.618,E2 -11675.618} C_VEL
LIN {X 0,Y 391.034,Z 400.662,A -85,B 0,C 180,E1 -11679.163,E2 -11679.163} C_VEL
LIN {X 0,Y 390.646,Z 405.858,A -85,B 0,C 180,E1 -11682.461,E2 -11682.461} C_VEL
LIN {X 0,Y 390.208,Z 412.661,A -85,B 0,C 180,E1 -11686.555,E2 -11686.555} C_VEL
LIN {X 0,Y 390.157,Z 413.599,A -85,B 0,C 180,E1 -11687.106,E2 -11687.106} C_VEL
LIN {X 0,Y 392.714,Z 424.312,A -85,B 0,C 180,E1 -11687.992,E2 -11687.992} C_VEL
LIN {X 0,Y 393.779,Z 431.552,A -85,B 0,C 180,E1 -11688.678,E2 -11688.678} C_VEL
LIN {X 0,Y 392.979,Z 441.515,A -85,B 0,C 180,E1 -11689.698,E2 -11689.698} C_VEL
LIN {X 0,Y 392.233,Z 449.285,A -85,B 0,C 180,E1 -11690.72,E2 -11690.72} C_VEL
LIN {X 0,Y 391.46,Z 456.919,A -85,B 0,C 180,E1 -11692.002,E2 -11692.002} C_VEL
LIN {X 0,Y 390.899,Z 462.777,A -85,B 0,C 180,E1 -11693.289,E2 -11693.289} C_VEL
LIN {X 0,Y 390.438,Z 466.442,A -85,B 0,C 180,E1 -11694.318,E2 -11694.318} C_VEL
LIN {X 0,Y 390.125,Z 469.276,A -85,B 0,C 180,E1 -11695.35,E2 -11695.35} C_VEL
LIN {X 0,Y 389.489,Z 472.191,A -85,B 0,C 180,E1 -11696.897,E2 -11696.897} C_VEL
LIN {X 0,Y 389.273,Z 473.259,A -85,B 0,C 180,E1 -11697.931,E2 -11697.931} C_VEL
LIN {X 0,Y 389.14,Z 473.662,A -85,B 0,C 180,E1 -11698.965,E2 -11698.965} C_VEL
LIN {X 0,Y 389.075,Z 473.403,A -85,B 0,C 180,E1 -11700,E2 -11700} C_VEL
LIN {X 0,Y 389.082,Z 472.475,A -85,B 0,C 180,E1 -11701.035,E2 -11701.035} C_VEL
LIN {X 0,Y 389.247,Z 469.799,A -85,B 0,C 180,E1 -11702.587,E2 -11702.587} C_VEL
LIN {X 0,Y 389.542,Z 465.476,A -85,B 0,C 180,E1 -11704.139,E2 -11704.139} C_VEL
LIN {X 0,Y 389.786,Z 460.429,A -85,B 0,C 180,E1 -11705.432,E2 -11705.432} C_VEL
LIN {X 0,Y 389.978,Z 453.818,A -85,B 0,C 180,E1 -11706.727,E2 -11706.727} C_VEL
LIN {X 0,Y 390.192,Z 446.5,A -85,B 0,C 180,E1 -11707.844,E2 -11707.844} C_VEL
LIN {X 0,Y 390.575,Z 437.384,A -85,B 0,C 180,E1 -11708.928,E2 -11708.928} C_VEL
LIN {X 0,Y 391.04,Z 427.431,A -85,B 0,C 180,E1 -11709.831,E2 -11709.831} C_VEL
LIN {X 0,Y 390.78,Z 422.128,A -85,B 0,C 180,E1 -11710.23,E2 -11710.23} C_VEL
LIN {X 0,Y 389.343,Z 411.858,A -85,B 0,C 180,E1 -11710.86,E2 -11710.86} C_VEL
LIN {X 0,Y 389.107,Z 409.49,A -85,B 0,C 180,E1 -11710.998,E2 -11710.998} C_VEL
LIN {X 0,Y 389.249,Z 403.426,A -85,B 0,C 180,E1 -11714.108,E2 -11714.108} C_VEL
LIN {X 0,Y 389.418,Z 397.958,A -85,B 0,C 180,E1 -11716.958,E2 -11716.958} C_VEL
LIN {X 0,Y 389.617,Z 391.692,A -85,B 0,C 180,E1 -11720.283,E2 -11720.283} C_VEL
LIN {X 0,Y 389.823,Z 384.916,A -85,B 0,C 180,E1 -11723.932,E2 -11723.932} C_VEL
LIN {X 0,Y 390.084,Z 378.68,A -85,B 0,C 180,E1 -11727.35,E2 -11727.35} C_VEL
LIN {X 0,Y 390.355,Z 373.445,A -85,B 0,C 180,E1 -11730.273,E2 -11730.273} C_VEL
LIN {X 0,Y 390.253,Z 371.877,A -85,B 0,C 180,E1 -11731.182,E2 -11731.182} C_VEL
LIN {X 0,Y 390.089,Z 371.894,A -85,B 0,C 180,E1 -11735.207,E2 -11735.207} C_VEL
LIN {X 0,Y 390.095,Z 371.895,A -85,B 0,C 180,E1 -11739.092,E2 -11739.092} C_VEL
LIN {X 0,Y 390.045,Z 371.899,A -85,B 0,C 180,E1 -11742.374,E2 -11742.374} C_VEL
LIN {X 0,Y 390.05,Z 371.898,A -85,B 0,C 180,E1 -11745.355,E2 -11745.355} C_VEL
LIN {X 0,Y 390.036,Z 371.901,A -85,B 0,C 180,E1 -11748.187,E2 -11748.187} C_VEL
LIN {X 0,Y 390.093,Z 371.896,A -85,B 0,C 180,E1 -11750.908,E2 -11750.908} C_VEL
LIN {X 0,Y 390.088,Z 371.895,A -85,B 0,C 180,E1 -11754.793,E2 -11754.793} C_VEL
LIN {X 0,Y 390.027,Z 371.903,A -85,B 0,C 180,E1 -11758.496,E2 -11758.496} C_VEL
LIN {X 0,Y 390.12,Z 371.891,A -85,B 0,C 180,E1 -11762.07,E2 -11762.07} C_VEL
LIN {X 0,Y 390.083,Z 371.892,A -85,B 0,C 180,E1 -11765.519,E2 -11765.519} C_VEL
LIN {X 0,Y 390.059,Z 371.898,A -85,B 0,C 180,E1 -11768.878,E2 -11768.878} C_VEL
LIN {X 0,Y 390.132,Z 371.89,A -85,B 0,C 180,E1 -11772.167,E2 -11772.167} C_VEL
LIN {X 0,Y 390.148,Z 371.884,A -85,B 0,C 180,E1 -11775.393,E2 -11775.393} C_VEL
LIN {X 0,Y 390.152,Z 371.886,A -85,B 0,C 180,E1 -11778.571,E2 -11778.571} C_VEL
LIN {X 0,Y 390.311,Z 371.868,A -85,B 0,C 180,E1 -11782.032,E2 -11782.032} C_VEL
LIN {X 0,Y 390.229,Z 371.875,A -85,B 0,C 180,E1 -11784.833,E2 -11784.833} C_VEL
LIN {X 0,Y 390.422,Z 371.855,A -85,B 0,C 180,E1 -11787.937,E2 -11787.937} C_VEL
LIN {X 0,Y 390.552,Z 371.838,A -85,B 0,C 180,E1 -11790,E2 -11790} C_VEL
LIN {X 0,Y 390.318,Z 371.864,A -85,B 0,C 180,E1 -11793.096,E2 -11793.096} C_VEL
LIN {X 0,Y 390.328,Z 371.865,A -85,B 0,C 180,E1 -11796.202,E2 -11796.202} C_VEL
LIN {X 0,Y 390.212,Z 371.877,A -85,B 0,C 180,E1 -11799.329,E2 -11799.329} C_VEL
LIN {X 0,Y 390.198,Z 371.882,A -85,B 0,C 180,E1 -11803.438,E2 -11803.438} C_VEL
LIN {X 0,Y 390.152,Z 371.886,A -85,B 0,C 180,E1 -11807.308,E2 -11807.308} C_VEL
LIN {X 0,Y 390.105,Z 371.89,A -85,B 0,C 180,E1 -11810.476,E2 -11810.476} C_VEL
LIN {X 0,Y 390.092,Z 371.896,A -85,B 0,C 180,E1 -11813.351,E2 -11813.351} C_VEL
LIN {X 0,Y 390.116,Z 371.889,A -85,B 0,C 180,E1 -11816.768,E2 -11816.768} C_VEL
LIN {X 0,Y 390.043,Z 371.897,A -85,B 0,C 180,E1 -11819.975,E2 -11819.975} C_VEL
LIN {X 0,Y 389.4,Z 371.979,A -85,B 0,C 180,E1 -11820.836,E2 -11820.836} C_VEL
LIN {X 0,Y 386.553,Z 372.334,A -85,B 0,C 180,E1 -11822.237,E2 -11822.237} C_VEL
LIN {X 0,Y 384.133,Z 372.638,A -85,B 0,C 180,E1 -11823.369,E2 -11823.369} C_VEL
LIN {X 0,Y 383.099,Z 372.763,A -85,B 0,C 180,E1 -11824.244,E2 -11824.244} C_VEL
LIN {X 0,Y 383.019,Z 372.773,A -85,B 0,C 180,E1 -11824.541,E2 -11824.541} C_VEL
LIN {X 0,Y 383.003,Z 372.776,A -85,B 0,C 180,E1 -11827.904,E2 -11827.904} C_VEL
LIN {X 0,Y 382.987,Z 372.782,A -85,B 0,C 180,E1 -11831.347,E2 -11831.347} C_VEL
LIN {X 0,Y 382.998,Z 372.775,A -85,B 0,C 180,E1 -11834.303,E2 -11834.303} C_VEL
LIN {X 0,Y 383.012,Z 372.777,A -85,B 0,C 180,E1 -11837.24,E2 -11837.24} C_VEL
LIN {X 0,Y 383.017,Z 372.773,A -85,B 0,C 180,E1 -11840.413,E2 -11840.413} C_VEL
LIN {X 0,Y 383.027,Z 372.771,A -85,B 0,C 180,E1 -11844.044,E2 -11844.044} C_VEL
LIN {X 0,Y 382.989,Z 372.778,A -85,B 0,C 180,E1 -11847.578,E2 -11847.578} C_VEL
LIN {X 0,Y 382.994,Z 372.777,A -85,B 0,C 180,E1 -11850.3,E2 -11850.3} C_VEL
LIN {X 0,Y 383.059,Z 372.77,A -85,B 0,C 180,E1 -11852.698,E2 -11852.698} C_VEL
LIN {X 0,Y 383.055,Z 372.772,A -85,B 0,C 180,E1 -11855.04,E2 -11855.04} C_VEL
LIN {X 0,Y 382.996,Z 372.778,A -85,B 0,C 180,E1 -11858.469,E2 -11858.469} C_VEL
LIN {X 0,Y 383.065,Z 372.767,A -85,B 0,C 180,E1 -11861.826,E2 -11861.826} C_VEL
LIN {X 0,Y 383.115,Z 372.762,A -85,B 0,C 180,E1 -11865.118,E2 -11865.118} C_VEL
LIN {X 0,Y 383.11,Z 372.764,A -85,B 0,C 180,E1 -11868.358,E2 -11868.358} C_VEL
LIN {X 0,Y 383.306,Z 372.738,A -85,B 0,C 180,E1 -11871.932,E2 -11871.932} C_VEL
LIN {X 0,Y 383.201,Z 372.754,A -85,B 0,C 180,E1 -11874.738,E2 -11874.738} C_VEL
LIN {X 0,Y 383.388,Z 372.727,A -85,B 0,C 180,E1 -11877.899,E2 -11877.899} C_VEL
LIN {X 0,Y 383.522,Z 372.712,A -85,B 0,C 180,E1 -11880,E2 -11880} C_VEL
LIN {X 0,Y 383.254,Z 372.744,A -85,B 0,C 180,E1 -11883.154,E2 -11883.154} C_VEL
LIN {X 0,Y 383.29,Z 372.743,A -85,B 0,C 180,E1 -11886.316,E2 -11886.316} C_VEL
LIN {X 0,Y 383.262,Z 372.746,A -85,B 0,C 180,E1 -11888.436,E2 -11888.436} C_VEL
LIN {X 0,Y 383.1,Z 372.764,A -85,B 0,C 180,E1 -11891.642,E2 -11891.642} C_VEL
LIN {X 0,Y 383.112,Z 372.762,A -85,B 0,C 180,E1 -11894.882,E2 -11894.882} C_VEL
LIN {X 0,Y 383.09,Z 372.769,A -85,B 0,C 180,E1 -11898.172,E2 -11898.172} C_VEL
LIN {X 0,Y 382.995,Z 372.777,A -85,B 0,C 180,E1 -11901.531,E2 -11901.531} C_VEL
LIN {X 0,Y 383.054,Z 372.769,A -85,B 0,C 180,E1 -11904.96,E2 -11904.96} C_VEL
LIN {X 0,Y 383.019,Z 372.773,A -85,B 0,C 180,E1 -11908.494,E2 -11908.494} C_VEL
LIN {X 0,Y 383.011,Z 372.777,A -85,B 0,C 180,E1 -11912.15,E2 -11912.15} C_VEL
LIN {X 0,Y 383.02,Z 372.773,A -85,B 0,C 180,E1 -11914.668,E2 -11914.668} C_VEL
LIN {X 0,Y 383.004,Z 372.779,A -85,B 0,C 180,E1 -11917.904,E2 -11917.904} C_VEL
LIN {X 0,Y 382.999,Z 372.776,A -85,B 0,C 180,E1 -11921.345,E2 -11921.345} C_VEL
LIN {X 0,Y 383.001,Z 372.777,A -85,B 0,C 180,E1 -11924.304,E2 -11924.304} C_VEL
LIN {X 0,Y 383.011,Z 372.776,A -85,B 0,C 180,E1 -11927.24,E2 -11927.24} C_VEL
LIN {X 0,Y 383.015,Z 372.771,A -85,B 0,C 180,E1 -11930.414,E2 -11930.414} C_VEL
LIN {X 0,Y 383.043,Z 372.927,A -85,B 0,C 180,E1 -11933.16,E2 -11933.16} C_VEL
LIN {X 0,Y 385.261,Z 383.407,A -85,B 0,C 180,E1 -11936.508,E2 -11936.508} C_VEL
LIN {X 0,Y 387.339,Z 393.103,A -85,B 0,C 180,E1 -11939.467,E2 -11939.467} C_VEL
LIN {X 0,Y 387.627,Z 397.358,A -85,B 0,C 180,E1 -11940.69,E2 -11940.69} C_VEL
LIN {X 0,Y 385.918,Z 410.888,A -85,B 0,C 180,E1 -11944.373,E2 -11944.373} C_VEL
LIN {X 0,Y 384.522,Z 424.396,A -85,B 0,C 180,E1 -11947.995,E2 -11947.995} C_VEL
LIN {X 0,Y 383.277,Z 440.485,A -85,B 0,C 180,E1 -11952.253,E2 -11952.253} C_VEL
LIN {X 0,Y 383.084,Z 442.757,A -85,B 0,C 180,E1 -11952.789,E2 -11952.789} C_VEL
LIN {X 0,Y 384.232,Z 456.673,A -85,B 0,C 180,E1 -11953.274,E2 -11953.274} C_VEL
LIN {X 0,Y 385.198,Z 469.002,A -85,B 0,C 180,E1 -11953.913,E2 -11953.913} C_VEL
LIN {X 0,Y 384.823,Z 479.911,A -85,B 0,C 180,E1 -11954.644,E2 -11954.644} C_VEL
LIN {X 0,Y 384.158,Z 491.166,A -85,B 0,C 180,E1 -11955.607,E2 -11955.607} C_VEL
LIN {X 0,Y 383.537,Z 501.787,A -85,B 0,C 180,E1 -11956.759,E2 -11956.759} C_VEL
LIN {X 0,Y 382.896,Z 511.563,A -85,B 0,C 180,E1 -11958.083,E2 -11958.083} C_VEL
LIN {X 0,Y 382.413,Z 519.531,A -85,B 0,C 180,E1 -11959.41,E2 -11959.41} C_VEL
LIN {X 0,Y 382.133,Z 527.229,A -85,B 0,C 180,E1 -11961.006,E2 -11961.006} C_VEL
LIN {X 0,Y 381.996,Z 533.328,A -85,B 0,C 180,E1 -11962.601,E2 -11962.601} C_VEL
LIN {X 0,Y 381.975,Z 538.072,A -85,B 0,C 180,E1 -11964.192,E2 -11964.192} C_VEL
LIN {X 0,Y 381.945,Z 541.595,A -85,B 0,C 180,E1 -11965.779,E2 -11965.779} C_VEL
LIN {X 0,Y 382.05,Z 543.325,A -85,B 0,C 180,E1 -11966.837,E2 -11966.837} C_VEL
LIN {X 0,Y 382.079,Z 544.585,A -85,B 0,C 180,E1 -11967.892,E2 -11967.892} C_VEL
LIN {X 0,Y 381.97,Z 545.406,A -85,B 0,C 180,E1 -11968.946,E2 -11968.946} C_VEL
LIN {X 0,Y 381.942,Z 545.762,A -85,B 0,C 180,E1 -11970,E2 -11970} C_VEL
LIN {X 0,Y 381.972,Z 545.693,A -85,B 0,C 180,E1 -11971.054,E2 -11971.054} C_VEL
LIN {X 0,Y 382.051,Z 545.216,A -85,B 0,C 180,E1 -11972.109,E2 -11972.109} C_VEL
LIN {X 0,Y 381.992,Z 544.266,A -85,B 0,C 180,E1 -11973.164,E2 -11973.164} C_VEL
LIN {X 0,Y 381.851,Z 542.865,A -85,B 0,C 180,E1 -11974.222,E2 -11974.222} C_VEL
LIN {X 0,Y 381.838,Z 539.529,A -85,B 0,C 180,E1 -11976.002,E2 -11976.002} C_VEL
LIN {X 0,Y 381.941,Z 535.942,A -85,B 0,C 180,E1 -11977.401,E2 -11977.401} C_VEL
LIN {X 0,Y 382.134,Z 529.779,A -85,B 0,C 180,E1 -11979.261,E2 -11979.261} C_VEL
LIN {X 0,Y 382.55,Z 523.008,A -85,B 0,C 180,E1 -11980.854,E2 -11980.854} C_VEL
LIN {X 0,Y 383.237,Z 514.623,A -85,B 0,C 180,E1 -11982.444,E2 -11982.444} C_VEL
LIN {X 0,Y 384.067,Z 504.815,A -85,B 0,C 180,E1 -11983.931,E2 -11983.931} C_VEL
LIN {X 0,Y 385.064,Z 494.334,A -85,B 0,C 180,E1 -11985.211,E2 -11985.211} C_VEL
LIN {X 0,Y 386.075,Z 483.591,A -85,B 0,C 180,E1 -11986.253,E2 -11986.253} C_VEL
LIN {X 0,Y 386.988,Z 472.364,A -85,B 0,C 180,E1 -11987.122,E2 -11987.122} C_VEL
LIN {X 0,Y 386.622,Z 460.045,A -85,B 0,C 180,E1 -11987.916,E2 -11987.916} C_VEL
LIN {X 0,Y 385.22,Z 447.529,A -85,B 0,C 180,E1 -11988.573,E2 -11988.573} C_VEL
LIN {X 0,Y 383.925,Z 440.676,A -85,B 0,C 180,E1 -11988.914,E2 -11988.914} C_VEL
LIN {X 0,Y 385.371,Z 427.764,A -85,B 0,C 180,E1 -11992.518,E2 -11992.518} C_VEL
LIN {X 0,Y 387.336,Z 414.922,A -85,B 0,C 180,E1 -11996.394,E2 -11996.394} C_VEL
LIN {X 0,Y 389.505,Z 405.156,A -85,B 0,C 180,E1 -11999.612,E2 -11999.612} C_VEL
LIN {X 0,Y 389.782,Z 403.272,A -85,B 0,C 180,E1 -12000.322,E2 -12000.322} C_VEL
LIN {X 0,Y 389.307,Z 399.446,A -85,B 0,C 180,E1 -12001.954,E2 -12001.954} C_VEL
LIN {X 0,Y 388.247,Z 393.861,A -85,B 0,C 180,E1 -12004.75,E2 -12004.75} C_VEL
LIN {X 0,Y 387.304,Z 390.213,A -85,B 0,C 180,E1 -12007.02,E2 -12007.02} C_VEL
LIN {X 0,Y 386.431,Z 386.272,A -85,B 0,C 180,E1 -12010.195,E2 -12010.195} C_VEL
LIN {X 0,Y 385.784,Z 383.908,A -85,B 0,C 180,E1 -12013.223,E2 -12013.223} C_VEL
LIN {X 0,Y 385.473,Z 382.751,A -85,B 0,C 180,E1 -12016.146,E2 -12016.146} C_VEL
LIN {X 0,Y 385.388,Z 382.653,A -85,B 0,C 180,E1 -12018.966,E2 -12018.966} C_VEL
LIN {X 0,Y 385.447,Z 383.412,A -85,B 0,C 180,E1 -12021.689,E2 -12021.689} C_VEL
LIN {X 0,Y 385.692,Z 385.377,A -85,B 0,C 180,E1 -12025.083,E2 -12025.083} C_VEL
LIN {X 0,Y 385.88,Z 386.827,A -85,B 0,C 180,E1 -12026.908,E2 -12026.908} C_VEL
LIN {X 0,Y 385.866,Z 389.177,A -85,B 0,C 180,E1 -12029.337,E2 -12029.337} C_VEL
LIN {X 0,Y 385.44,Z 391.93,A -85,B 0,C 180,E1 -12031.701,E2 -12031.701} C_VEL
LIN {X 0,Y 384.763,Z 396.495,A -85,B 0,C 180,E1 -12035.158,E2 -12035.158} C_VEL
LIN {X 0,Y 384.13,Z 401.892,A -85,B 0,C 180,E1 -12038.922,E2 -12038.922} C_VEL
LIN {X 0,Y 383.703,Z 407.004,A -85,B 0,C 180,E1 -12042.26,E2 -12042.26} C_VEL
LIN {X 0,Y 383.206,Z 414.102,A -85,B 0,C 180,E1 -12046.635,E2 -12046.635} C_VEL
LIN {X 0,Y 385.783,Z 424.112,A -85,B 0,C 180,E1 -12047.506,E2 -12047.506} C_VEL
LIN {X 0,Y 387.125,Z 432.599,A -85,B 0,C 180,E1 -12048.348,E2 -12048.348} C_VEL
LIN {X 0,Y 386.354,Z 441.574,A -85,B 0,C 180,E1 -12049.281,E2 -12049.281} C_VEL
LIN {X 0,Y 385.603,Z 449.286,A -85,B 0,C 180,E1 -12050.294,E2 -12050.294} C_VEL
LIN {X 0,Y 384.719,Z 457.061,A -85,B 0,C 180,E1 -12051.597,E2 -12051.597} C_VEL
LIN {X 0,Y 384.061,Z 463.02,A -85,B 0,C 180,E1 -12052.905,E2 -12052.905} C_VEL
LIN {X 0,Y 383.468,Z 467.559,A -85,B 0,C 180,E1 -12054.215,E2 -12054.215} C_VEL
LIN {X 0,Y 382.818,Z 471.418,A -85,B 0,C 180,E1 -12055.789,E2 -12055.789} C_VEL
LIN {X 0,Y 382.458,Z 473.095,A -85,B 0,C 180,E1 -12056.84,E2 -12056.84} C_VEL
LIN {X 0,Y 382.227,Z 474.087,A -85,B 0,C 180,E1 -12057.893,E2 -12057.893} C_VEL
LIN {X 0,Y 382.085,Z 474.416,A -85,B 0,C 180,E1 -12058.946,E2 -12058.946} C_VEL
LIN {X 0,Y 382.018,Z 474.081,A -85,B 0,C 180,E1 -12060,E2 -12060} C_VEL
LIN {X 0,Y 382.03,Z 473.076,A -85,B 0,C 180,E1 -12061.054,E2 -12061.054} C_VEL
LIN {X 0,Y 382.199,Z 470.29,A -85,B 0,C 180,E1 -12062.635,E2 -12062.635} C_VEL
LIN {X 0,Y 382.495,Z 465.85,A -85,B 0,C 180,E1 -12064.215,E2 -12064.215} C_VEL
LIN {X 0,Y 382.719,Z 460.701,A -85,B 0,C 180,E1 -12065.532,E2 -12065.532} C_VEL
LIN {X 0,Y 382.943,Z 453.953,A -85,B 0,C 180,E1 -12066.851,E2 -12066.851} C_VEL
LIN {X 0,Y 383.134,Z 446.595,A -85,B 0,C 180,E1 -12067.976,E2 -12067.976} C_VEL
LIN {X 0,Y 383.564,Z 437.183,A -85,B 0,C 180,E1 -12069.093,E2 -12069.093} C_VEL
LIN {X 0,Y 384.029,Z 427.025,A -85,B 0,C 180,E1 -12070.012,E2 -12070.012} C_VEL
LIN {X 0,Y 383.305,Z 419.512,A -85,B 0,C 180,E1 -12070.565,E2 -12070.565} C_VEL
LIN {X 0,Y 382.059,Z 409.797,A -85,B 0,C 180,E1 -12071.137,E2 -12071.137} C_VEL
LIN {X 0,Y 382.185,Z 403.56,A -85,B 0,C 180,E1 -12074.374,E2 -12074.374} C_VEL
LIN {X 0,Y 382.383,Z 397.344,A -85,B 0,C 180,E1 -12077.654,E2 -12077.654} C_VEL
LIN {X 0,Y 382.572,Z 391.143,A -85,B 0,C 180,E1 -12080.991,E2 -12080.991} C_VEL
LIN {X 0,Y 382.804,Z 384.908,A -85,B 0,C 180,E1 -12084.399,E2 -12084.399} C_VEL
LIN {X 0,Y 383.045,Z 379.674,A -85,B 0,C 180,E1 -12087.303,E2 -12087.303} C_VEL
LIN {X 0,Y 383.304,Z 375.455,A -85,B 0,C 180,E1 -12089.674,E2 -12089.674} C_VEL
LIN {X 0,Y 383.198,Z 372.755,A -85,B 0,C 180,E1 -12091.283,E2 -12091.283} C_VEL
LIN {X 0,Y 383.021,Z 372.776,A -85,B 0,C 180,E1 -12094.668,E2 -12094.668} C_VEL
LIN {X 0,Y 383.005,Z 372.775,A -85,B 0,C 180,E1 -12097.904,E2 -12097.904} C_VEL
LIN {X 0,Y 382.987,Z 372.778,A -85,B 0,C 180,E1 -12101.347,E2 -12101.347} C_VEL
LIN {X 0,Y 383,Z 372.776,A -85,B 0,C 180,E1 -12104.304,E2 -12104.304} C_VEL
LIN {X 0,Y 383.013,Z 372.775,A -85,B 0,C 180,E1 -12107.24,E2 -12107.24} C_VEL
LIN {X 0,Y 383.018,Z 372.776,A -85,B 0,C 180,E1 -12110.414,E2 -12110.414} C_VEL
LIN {X 0,Y 383.028,Z 372.772,A -85,B 0,C 180,E1 -12114.045,E2 -12114.045} C_VEL
LIN {X 0,Y 382.99,Z 372.776,A -85,B 0,C 180,E1 -12117.578,E2 -12117.578} C_VEL
LIN {X 0,Y 382.996,Z 372.779,A -85,B 0,C 180,E1 -12120.3,E2 -12120.3} C_VEL
LIN {X 0,Y 383.083,Z 372.766,A -85,B 0,C 180,E1 -12124.021,E2 -12124.021} C_VEL
LIN {X 0,Y 383.011,Z 372.773,A -85,B 0,C 180,E1 -12127.335,E2 -12127.335} C_VEL
LIN {X 0,Y 383.064,Z 372.77,A -85,B 0,C 180,E1 -12130.716,E2 -12130.716} C_VEL
LIN {X 0,Y 383.084,Z 372.767,A -85,B 0,C 180,E1 -12134.027,E2 -12134.027} C_VEL
LIN {X 0,Y 383.14,Z 372.757,A -85,B 0,C 180,E1 -12137.284,E2 -12137.284} C_VEL
LIN {X 0,Y 383.155,Z 372.759,A -85,B 0,C 180,E1 -12140.498,E2 -12140.498} C_VEL
LIN {X 0,Y 383.284,Z 372.742,A -85,B 0,C 180,E1 -12143.684,E2 -12143.684} C_VEL
LIN {X 0,Y 383.389,Z 372.73,A -85,B 0,C 180,E1 -12147.899,E2 -12147.899} C_VEL
LIN {X 0,Y 383.521,Z 372.714,A -85,B 0,C 180,E1 -12150,E2 -12150} C_VEL
LIN {X 0,Y 383.254,Z 372.744,A -85,B 0,C 180,E1 -12153.154,E2 -12153.154} C_VEL
LIN {X 0,Y 383.284,Z 372.742,A -85,B 0,C 180,E1 -12156.316,E2 -12156.316} C_VEL
LIN {X 0,Y 383.158,Z 372.757,A -85,B 0,C 180,E1 -12159.502,E2 -12159.502} C_VEL
LIN {X 0,Y 383.128,Z 372.763,A -85,B 0,C 180,E1 -12163.536,E2 -12163.536} C_VEL
LIN {X 0,Y 383.099,Z 372.765,A -85,B 0,C 180,E1 -12167.455,E2 -12167.455} C_VEL
LIN {X 0,Y 383.047,Z 372.768,A -85,B 0,C 180,E1 -12170.653,E2 -12170.653} C_VEL
LIN {X 0,Y 383.036,Z 372.774,A -85,B 0,C 180,E1 -12173.807,E2 -12173.807} C_VEL
LIN {X 0,Y 383.083,Z 372.766,A -85,B 0,C 180,E1 -12176.123,E2 -12176.123} C_VEL
LIN {X 0,Y 382.995,Z 372.779,A -85,B 0,C 180,E1 -12179.7,E2 -12179.7} C_VEL
LIN {X 0,Y 383.006,Z 372.778,A -85,B 0,C 180,E1 -12183.401,E2 -12183.401} C_VEL
LIN {X 0,Y 383.019,Z 372.773,A -85,B 0,C 180,E1 -12184.541,E2 -12184.541} C_VEL
LIN {X 0,Y 382.355,Z 372.859,A -85,B 0,C 180,E1 -12185.417,E2 -12185.417} C_VEL
LIN {X 0,Y 379.481,Z 373.215,A -85,B 0,C 180,E1 -12186.842,E2 -12186.842} C_VEL
LIN {X 0,Y 377.054,Z 373.517,A -85,B 0,C 180,E1 -12187.994,E2 -12187.994} C_VEL
LIN {X 0,Y 376.028,Z 373.645,A -85,B 0,C 180,E1 -12188.885,E2 -12188.885} C_VEL
LIN {X 0,Y 375.954,Z 373.655,A -85,B 0,C 180,E1 -12189.187,E2 -12189.187} C_VEL
LIN {X 0,Y 375.934,Z 373.654,A -85,B 0,C 180,E1 -12192.3,E2 -12192.3} C_VEL
LIN {X 0,Y 375.929,Z 373.659,A -85,B 0,C 180,E1 -12195.268,E2 -12195.268} C_VEL
LIN {X 0,Y 375.936,Z 373.655,A -85,B 0,C 180,E1 -12198.399,E2 -12198.399} C_VEL
LIN {X 0,Y 375.976,Z 373.65,A -85,B 0,C 180,E1 -12201.729,E2 -12201.729} C_VEL
LIN {X 0,Y 375.982,Z 373.652,A -85,B 0,C 180,E1 -12205.333,E2 -12205.333} C_VEL
LIN {X 0,Y 375.96,Z 373.653,A -85,B 0,C 180,E1 -12208.438,E2 -12208.438} C_VEL
LIN {X 0,Y 375.998,Z 373.647,A -85,B 0,C 180,E1 -12212.141,E2 -12212.141} C_VEL
LIN {X 0,Y 376.009,Z 373.647,A -85,B 0,C 180,E1 -12214.539,E2 -12214.539} C_VEL
LIN {X 0,Y 375.966,Z 373.652,A -85,B 0,C 180,E1 -12218.046,E2 -12218.046} C_VEL
LIN {X 0,Y 376.011,Z 373.646,A -85,B 0,C 180,E1 -12221.473,E2 -12221.473} C_VEL
LIN {X 0,Y 376.062,Z 373.643,A -85,B 0,C 180,E1 -12224.833,E2 -12224.833} C_VEL
LIN {X 0,Y 376.061,Z 373.64,A -85,B 0,C 180,E1 -12228.137,E2 -12228.137} C_VEL
LIN {X 0,Y 376.26,Z 373.615,A -85,B 0,C 180,E1 -12231.877,E2 -12231.877} C_VEL
LIN {X 0,Y 376.173,Z 373.63,A -85,B 0,C 180,E1 -12234.64,E2 -12234.64} C_VEL
LIN {X 0,Y 376.354,Z 373.603,A -85,B 0,C 180,E1 -12237.86,E2 -12237.86} C_VEL
LIN {X 0,Y 376.492,Z 373.587,A -85,B 0,C 180,E1 -12240,E2 -12240} C_VEL
LIN {X 0,Y 376.192,Z 373.623,A -85,B 0,C 180,E1 -12243.213,E2 -12243.213} C_VEL
LIN {X 0,Y 376.249,Z 373.621,A -85,B 0,C 180,E1 -12246.435,E2 -12246.435} C_VEL
LIN {X 0,Y 376.207,Z 373.624,A -85,B 0,C 180,E1 -12248.595,E2 -12248.595} C_VEL
LIN {X 0,Y 376.052,Z 373.643,A -85,B 0,C 180,E1 -12251.863,E2 -12251.863} C_VEL
LIN {X 0,Y 376.06,Z 373.639,A -85,B 0,C 180,E1 -12255.167,E2 -12255.167} C_VEL
LIN {X 0,Y 376.025,Z 373.646,A -85,B 0,C 180,E1 -12258.526,E2 -12258.526} C_VEL
LIN {X 0,Y 375.965,Z 373.656,A -85,B 0,C 180,E1 -12261.954,E2 -12261.954} C_VEL
LIN {X 0,Y 376.008,Z 373.647,A -85,B 0,C 180,E1 -12265.461,E2 -12265.461} C_VEL
LIN {X 0,Y 375.962,Z 373.65,A -85,B 0,C 180,E1 -12269.08,E2 -12269.08} C_VEL
LIN {X 0,Y 375.952,Z 373.653,A -85,B 0,C 180,E1 -12272.828,E2 -12272.828} C_VEL
LIN {X 0,Y 375.96,Z 373.654,A -85,B 0,C 180,E1 -12275.415,E2 -12275.415} C_VEL
LIN {X 0,Y 375.978,Z 373.651,A -85,B 0,C 180,E1 -12278.271,E2 -12278.271} C_VEL
LIN {X 0,Y 375.946,Z 373.657,A -85,B 0,C 180,E1 -12281.603,E2 -12281.603} C_VEL
LIN {X 0,Y 375.957,Z 373.654,A -85,B 0,C 180,E1 -12285.264,E2 -12285.264} C_VEL
LIN {X 0,Y 375.942,Z 373.655,A -85,B 0,C 180,E1 -12289.133,E2 -12289.133} C_VEL
LIN {X 0,Y 376.018,Z 373.772,A -85,B 0,C 180,E1 -12292.805,E2 -12292.805} C_VEL
LIN {X 0,Y 378.493,Z 385.601,A -85,B 0,C 180,E1 -12296.676,E2 -12296.676} C_VEL
LIN {X 0,Y 380.554,Z 395.663,A -85,B 0,C 180,E1 -12299.785,E2 -12299.785} C_VEL
LIN {X 0,Y 380.534,Z 398.963,A -85,B 0,C 180,E1 -12300.738,E2 -12300.738} C_VEL
LIN {X 0,Y 378.96,Z 411.267,A -85,B 0,C 180,E1 -12304.163,E2 -12304.163} C_VEL
LIN {X 0,Y 377.381,Z 425.726,A -85,B 0,C 180,E1 -12308.133,E2 -12308.133} C_VEL
LIN {X 0,Y 376.147,Z 441.26,A -85,B 0,C 180,E1 -12312.344,E2 -12312.344} C_VEL
LIN {X 0,Y 376.025,Z 442.216,A -85,B 0,C 180,E1 -12312.6,E2 -12312.6} C_VEL
LIN {X 0,Y 377.121,Z 455.903,A -85,B 0,C 180,E1 -12313.088,E2 -12313.088} C_VEL
LIN {X 0,Y 378.05,Z 468.312,A -85,B 0,C 180,E1 -12313.739,E2 -12313.739} C_VEL
LIN {X 0,Y 377.879,Z 477.55,A -85,B 0,C 180,E1 -12314.355,E2 -12314.355} C_VEL
LIN {X 0,Y 377.268,Z 488.739,A -85,B 0,C 180,E1 -12315.297,E2 -12315.297} C_VEL
LIN {X 0,Y 376.521,Z 498.685,A -85,B 0,C 180,E1 -12316.343,E2 -12316.343} C_VEL
LIN {X 0,Y 376.091,Z 506.322,A -85,B 0,C 180,E1 -12317.316,E2 -12317.316} C_VEL
LIN {X 0,Y 375.604,Z 515.151,A -85,B 0,C 180,E1 -12318.67,E2 -12318.67} C_VEL
LIN {X 0,Y 375.199,Z 522.365,A -85,B 0,C 180,E1 -12320.022,E2 -12320.022} C_VEL
LIN {X 0,Y 375.011,Z 529.343,A -85,B 0,C 180,E1 -12321.649,E2 -12321.649} C_VEL
LIN {X 0,Y 374.884,Z 535.637,A -85,B 0,C 180,E1 -12323.542,E2 -12323.542} C_VEL
LIN {X 0,Y 374.829,Z 539.626,A -85,B 0,C 180,E1 -12325.16,E2 -12325.16} C_VEL
LIN {X 0,Y 374.981,Z 542.484,A -85,B 0,C 180,E1 -12326.777,E2 -12326.777} C_VEL
LIN {X 0,Y 375.032,Z 543.775,A -85,B 0,C 180,E1 -12327.852,E2 -12327.852} C_VEL
LIN {X 0,Y 374.922,Z 544.624,A -85,B 0,C 180,E1 -12328.926,E2 -12328.926} C_VEL
LIN {X 0,Y 374.891,Z 545.037,A -85,B 0,C 180,E1 -12330,E2 -12330} C_VEL
LIN {X 0,Y 374.923,Z 544.994,A -85,B 0,C 180,E1 -12331.074,E2 -12331.074} C_VEL
LIN {X 0,Y 374.986,Z 544.54,A -85,B 0,C 180,E1 -12332.148,E2 -12332.148} C_VEL
LIN {X 0,Y 374.923,Z 543.644,A -85,B 0,C 180,E1 -12333.224,E2 -12333.224} C_VEL
LIN {X 0,Y 374.768,Z 542.266,A -85,B 0,C 180,E1 -12334.302,E2 -12334.302} C_VEL
LIN {X 0,Y 374.745,Z 539.309,A -85,B 0,C 180,E1 -12335.962,E2 -12335.962} C_VEL
LIN {X 0,Y 374.86,Z 535.457,A -85,B 0,C 180,E1 -12337.541,E2 -12337.541} C_VEL
LIN {X 0,Y 375.01,Z 530.342,A -85,B 0,C 180,E1 -12339.166,E2 -12339.166} C_VEL
LIN {X 0,Y 375.395,Z 523.938,A -85,B 0,C 180,E1 -12340.79,E2 -12340.79} C_VEL
LIN {X 0,Y 376.129,Z 515.927,A -85,B 0,C 180,E1 -12342.409,E2 -12342.409} C_VEL
LIN {X 0,Y 377.048,Z 505.995,A -85,B 0,C 180,E1 -12344.023,E2 -12344.023} C_VEL
LIN {X 0,Y 378.107,Z 495.634,A -85,B 0,C 180,E1 -12345.359,E2 -12345.359} C_VEL
LIN {X 0,Y 379.155,Z 485.459,A -85,B 0,C 180,E1 -12346.42,E2 -12346.42} C_VEL
LIN {X 0,Y 380.162,Z 474.658,A -85,B 0,C 180,E1 -12347.324,E2 -12347.324} C_VEL
LIN {X 0,Y 380.015,Z 461.317,A -85,B 0,C 180,E1 -12348.246,E2 -12348.246} C_VEL
LIN {X 0,Y 378.743,Z 449.22,A -85,B 0,C 180,E1 -12348.935,E2 -12348.935} C_VEL
LIN {X 0,Y 377.094,Z 440.354,A -85,B 0,C 180,E1 -12349.389,E2 -12349.389} C_VEL
LIN {X 0,Y 378.566,Z 428.017,A -85,B 0,C 180,E1 -12352.946,E2 -12352.946} C_VEL
LIN {X 0,Y 380.697,Z 415.414,A -85,B 0,C 180,E1 -12356.891,E2 -12356.891} C_VEL
LIN {X 0,Y 382.7,Z 407.113,A -85,B 0,C 180,E1 -12359.725,E2 -12359.725} C_VEL
LIN {X 0,Y 383.004,Z 405.277,A -85,B 0,C 180,E1 -12360.409,E2 -12360.409} C_VEL
LIN {X 0,Y 382.296,Z 399.901,A -85,B 0,C 180,E1 -12362.841,E2 -12362.841} C_VEL
LIN {X 0,Y 381.548,Z 396.162,A -85,B 0,C 180,E1 -12364.821,E2 -12364.821} C_VEL
LIN {X 0,Y 380.497,Z 392.014,A -85,B 0,C 180,E1 -12367.556,E2 -12367.556} C_VEL
LIN {X 0,Y 379.771,Z 388.667,A -85,B 0,C 180,E1 -12370.369,E2 -12370.369} C_VEL
LIN {X 0,Y 379.172,Z 386.424,A -85,B 0,C 180,E1 -12373.299,E2 -12373.299} C_VEL
LIN {X 0,Y 378.834,Z 385.237,A -85,B 0,C 180,E1 -12376.346,E2 -12376.346} C_VEL
LIN {X 0,Y 378.706,Z 385.194,A -85,B 0,C 180,E1 -12379.542,E2 -12379.542} C_VEL
LIN {X 0,Y 378.741,Z 386.006,A -85,B 0,C 180,E1 -12382.24,E2 -12382.24} C_VEL
LIN {X 0,Y 378.926,Z 387.457,A -85,B 0,C 180,E1 -12384.903,E2 -12384.903} C_VEL
LIN {X 0,Y 379.093,Z 389.462,A -85,B 0,C 180,E1 -12387.477,E2 -12387.477} C_VEL
LIN {X 0,Y 379.103,Z 390.594,A -85,B 0,C 180,E1 -12388.73,E2 -12388.73} C_VEL
LIN {X 0,Y 378.728,Z 393.247,A -85,B 0,C 180,E1 -12391.153,E2 -12391.153} C_VEL
LIN {X 0,Y 377.952,Z 397.632,A -85,B 0,C 180,E1 -12394.679,E2 -12394.679} C_VEL
LIN {X 0,Y 377.31,Z 402.382,A -85,B 0,C 180,E1 -12398.128,E2 -12398.128} C_VEL
LIN {X 0,Y 376.806,Z 408.162,A -85,B 0,C 180,E1 -12402.033,E2 -12402.033} C_VEL
LIN {X 0,Y 376.273,Z 414.666,A -85,B 0,C 180,E1 -12406.134,E2 -12406.134} C_VEL
LIN {X 0,Y 379.163,Z 425.688,A -85,B 0,C 180,E1 -12407.148,E2 -12407.148} C_VEL
LIN {X 0,Y 380.505,Z 433.904,A -85,B 0,C 180,E1 -12408.007,E2 -12408.007} C_VEL
LIN {X 0,Y 379.598,Z 443.499,A -85,B 0,C 180,E1 -12409.06,E2 -12409.06} C_VEL
LIN {X 0,Y 378.801,Z 450.856,A -85,B 0,C 180,E1 -12410.087,E2 -12410.087} C_VEL
LIN {X 0,Y 377.84,Z 458.593,A -85,B 0,C 180,E1 -12411.442,E2 -12411.442} C_VEL
LIN {X 0,Y 377.158,Z 464.364,A -85,B 0,C 180,E1 -12412.774,E2 -12412.774} C_VEL
LIN {X 0,Y 376.499,Z 468.746,A -85,B 0,C 180,E1 -12414.107,E2 -12414.107} C_VEL
LIN {X 0,Y 375.809,Z 472.428,A -85,B 0,C 180,E1 -12415.71,E2 -12415.71} C_VEL
LIN {X 0,Y 375.428,Z 474.002,A -85,B 0,C 180,E1 -12416.781,E2 -12416.781} C_VEL
LIN {X 0,Y 375.179,Z 474.904,A -85,B 0,C 180,E1 -12417.853,E2 -12417.853} C_VEL
LIN {X 0,Y 375.031,Z 475.154,A -85,B 0,C 180,E1 -12418.926,E2 -12418.926} C_VEL
LIN {X 0,Y 374.964,Z 474.738,A -85,B 0,C 180,E1 -12420,E2 -12420} C_VEL
LIN {X 0,Y 374.978,Z 473.651,A -85,B 0,C 180,E1 -12421.074,E2 -12421.074} C_VEL
LIN {X 0,Y 375.135,Z 470.734,A -85,B 0,C 180,E1 -12422.685,E2 -12422.685} C_VEL
LIN {X 0,Y 375.432,Z 466.151,A -85,B 0,C 180,E1 -12424.294,E2 -12424.294} C_VEL
LIN {X 0,Y 375.65,Z 460.892,A -85,B 0,C 180,E1 -12425.637,E2 -12425.637} C_VEL
LIN {X 0,Y 375.892,Z 454.019,A -85,B 0,C 180,E1 -12426.98,E2 -12426.98} C_VEL
LIN {X 0,Y 376.087,Z 446.95,A -85,B 0,C 180,E1 -12428.072,E2 -12428.072} C_VEL
LIN {X 0,Y 376.493,Z 438.263,A -85,B 0,C 180,E1 -12429.13,E2 -12429.13} C_VEL
LIN {X 0,Y 376.966,Z 428.28,A -85,B 0,C 180,E1 -12430.066,E2 -12430.066} C_VEL
LIN {X 0,Y 376.378,Z 420.961,A -85,B 0,C 180,E1 -12430.626,E2 -12430.626} C_VEL
LIN {X 0,Y 375.007,Z 410.091,A -85,B 0,C 180,E1 -12431.28,E2 -12431.28} C_VEL
LIN {X 0,Y 375.103,Z 404.72,A -85,B 0,C 180,E1 -12434.098,E2 -12434.098} C_VEL
LIN {X 0,Y 375.309,Z 398.466,A -85,B 0,C 180,E1 -12437.435,E2 -12437.435} C_VEL
LIN {X 0,Y 375.52,Z 392.215,A -85,B 0,C 180,E1 -12440.83,E2 -12440.83} C_VEL
LIN {X 0,Y 375.746,Z 385.93,A -85,B 0,C 180,E1 -12444.299,E2 -12444.299} C_VEL
LIN {X 0,Y 376.036,Z 379.614,A -85,B 0,C 180,E1 -12447.856,E2 -12447.856} C_VEL
LIN {X 0,Y 376.261,Z 375.354,A -85,B 0,C 180,E1 -12450.286,E2 -12450.286} C_VEL
LIN {X 0,Y 376.148,Z 373.633,A -85,B 0,C 180,E1 -12451.328,E2 -12451.328} C_VEL
LIN {X 0,Y 375.961,Z 373.653,A -85,B 0,C 180,E1 -12455.415,E2 -12455.415} C_VEL
LIN {X 0,Y 375.979,Z 373.651,A -85,B 0,C 180,E1 -12458.271,E2 -12458.271} C_VEL
LIN {X 0,Y 375.937,Z 373.655,A -85,B 0,C 180,E1 -12461.601,E2 -12461.601} C_VEL
LIN {X 0,Y 375.957,Z 373.653,A -85,B 0,C 180,E1 -12465.264,E2 -12465.264} C_VEL
LIN {X 0,Y 375.944,Z 373.656,A -85,B 0,C 180,E1 -12469.133,E2 -12469.133} C_VEL
LIN {X 0,Y 375.967,Z 373.652,A -85,B 0,C 180,E1 -12471.912,E2 -12471.912} C_VEL
LIN {X 0,Y 375.983,Z 373.649,A -85,B 0,C 180,E1 -12475.333,E2 -12475.333} C_VEL
LIN {X 0,Y 375.961,Z 373.656,A -85,B 0,C 180,E1 -12478.438,E2 -12478.438} C_VEL
LIN {X 0,Y 375.987,Z 373.652,A -85,B 0,C 180,E1 -12482.14,E2 -12482.14} C_VEL
LIN {X 0,Y 376.01,Z 373.65,A -85,B 0,C 180,E1 -12484.539,E2 -12484.539} C_VEL
LIN {X 0,Y 375.966,Z 373.654,A -85,B 0,C 180,E1 -12488.046,E2 -12488.046} C_VEL
LIN {X 0,Y 376.027,Z 373.644,A -85,B 0,C 180,E1 -12491.474,E2 -12491.474} C_VEL
LIN {X 0,Y 376.062,Z 373.64,A -85,B 0,C 180,E1 -12494.833,E2 -12494.833} C_VEL
LIN {X 0,Y 376.054,Z 373.645,A -85,B 0,C 180,E1 -12498.137,E2 -12498.137} C_VEL
LIN {X 0,Y 376.222,Z 373.623,A -85,B 0,C 180,E1 -12501.919,E2 -12501.919} C_VEL
LIN {X 0,Y 376.173,Z 373.627,A -85,B 0,C 180,E1 -12504.64,E2 -12504.64} C_VEL
LIN {X 0,Y 376.355,Z 373.606,A -85,B 0,C 180,E1 -12507.86,E2 -12507.86} C_VEL
LIN {X 0,Y 376.491,Z 373.59,A -85,B 0,C 180,E1 -12510,E2 -12510} C_VEL
LIN {X 0,Y 376.192,Z 373.624,A -85,B 0,C 180,E1 -12513.213,E2 -12513.213} C_VEL
LIN {X 0,Y 376.242,Z 373.618,A -85,B 0,C 180,E1 -12516.435,E2 -12516.435} C_VEL
LIN {X 0,Y 376.125,Z 373.635,A -85,B 0,C 180,E1 -12519.681,E2 -12519.681} C_VEL
LIN {X 0,Y 376.092,Z 373.639,A -85,B 0,C 180,E1 -12523.658,E2 -12523.658} C_VEL
LIN {X 0,Y 376.048,Z 373.644,A -85,B 0,C 180,E1 -12527.608,E2 -12527.608} C_VEL
LIN {X 0,Y 376.009,Z 373.645,A -85,B 0,C 180,E1 -12530.843,E2 -12530.843} C_VEL
LIN {X 0,Y 375.997,Z 373.648,A -85,B 0,C 180,E1 -12534.281,E2 -12534.281} C_VEL
LIN {X 0,Y 376.022,Z 373.644,A -85,B 0,C 180,E1 -12536.652,E2 -12536.652} C_VEL
LIN {X 0,Y 375.967,Z 373.65,A -85,B 0,C 180,E1 -12540.312,E2 -12540.312} C_VEL
LIN {X 0,Y 375.962,Z 373.652,A -85,B 0,C 180,E1 -12544.111,E2 -12544.111} C_VEL
LIN {X 0,Y 375.956,Z 373.653,A -85,B 0,C 180,E1 -12546.741,E2 -12546.741} C_VEL
LIN {X 0,Y 375.954,Z 373.655,A -85,B 0,C 180,E1 -12549.187,E2 -12549.187} C_VEL
LIN {X 0,Y 375.31,Z 373.741,A -85,B 0,C 180,E1 -12550.08,E2 -12550.08} C_VEL
LIN {X 0,Y 372.458,Z 374.098,A -85,B 0,C 180,E1 -12551.533,E2 -12551.533} C_VEL
LIN {X 0,Y 370.019,Z 374.398,A -85,B 0,C 180,E1 -12552.708,E2 -12552.708} C_VEL
LIN {X 0,Y 368.96,Z 374.526,A -85,B 0,C 180,E1 -12553.617,E2 -12553.617} C_VEL
LIN {X 0,Y 368.868,Z 374.535,A -85,B 0,C 180,E1 -12553.925,E2 -12553.925} C_VEL
LIN {X 0,Y 368.887,Z 374.534,A -85,B 0,C 180,E1 -12556.696,E2 -12556.696} C_VEL
LIN {X 0,Y 368.913,Z 374.531,A -85,B 0,C 180,E1 -12559.643,E2 -12559.643} C_VEL
LIN {X 0,Y 368.903,Z 374.535,A -85,B 0,C 180,E1 -12563.144,E2 -12563.144} C_VEL
LIN {X 0,Y 368.898,Z 374.532,A -85,B 0,C 180,E1 -12566.462,E2 -12566.462} C_VEL
LIN {X 0,Y 368.931,Z 374.531,A -85,B 0,C 180,E1 -12569.046,E2 -12569.046} C_VEL
LIN {X 0,Y 368.982,Z 374.522,A -85,B 0,C 180,E1 -12571.564,E2 -12571.564} C_VEL
LIN {X 0,Y 369.002,Z 374.517,A -85,B 0,C 180,E1 -12574.02,E2 -12574.02} C_VEL
LIN {X 0,Y 368.935,Z 374.527,A -85,B 0,C 180,E1 -12577.605,E2 -12577.605} C_VEL
LIN {X 0,Y 368.961,Z 374.527,A -85,B 0,C 180,E1 -12581.106,E2 -12581.106} C_VEL
LIN {X 0,Y 369.001,Z 374.521,A -85,B 0,C 180,E1 -12584.535,E2 -12584.535} C_VEL
LIN {X 0,Y 369.015,Z 374.517,A -85,B 0,C 180,E1 -12587.907,E2 -12587.907} C_VEL
LIN {X 0,Y 369.232,Z 374.49,A -85,B 0,C 180,E1 -12591.8,E2 -12591.8} C_VEL
LIN {X 0,Y 369.146,Z 374.505,A -85,B 0,C 180,E1 -12594.537,E2 -12594.537} C_VEL
LIN {X 0,Y 369.319,Z 374.479,A -85,B 0,C 180,E1 -12597.819,E2 -12597.819} C_VEL
LIN {X 0,Y 369.461,Z 374.463,A -85,B 0,C 180,E1 -12600,E2 -12600} C_VEL
LIN {X 0,Y 369.321,Z 374.482,A -85,B 0,C 180,E1 -12602.181,E2 -12602.181} C_VEL
LIN {X 0,Y 369.211,Z 374.496,A -85,B 0,C 180,E1 -12606.558,E2 -12606.558} C_VEL
LIN {X 0,Y 369.14,Z 374.504,A -85,B 0,C 180,E1 -12608.761,E2 -12608.761} C_VEL
LIN {X 0,Y 369.008,Z 374.522,A -85,B 0,C 180,E1 -12612.093,E2 -12612.093} C_VEL
LIN {X 0,Y 369,Z 374.519,A -85,B 0,C 180,E1 -12615.465,E2 -12615.465} C_VEL
LIN {X 0,Y 368.984,Z 374.521,A -85,B 0,C 180,E1 -12618.893,E2 -12618.893} C_VEL
LIN {X 0,Y 368.934,Z 374.531,A -85,B 0,C 180,E1 -12622.395,E2 -12622.395} C_VEL
LIN {X 0,Y 369.002,Z 374.522,A -85,B 0,C 180,E1 -12625.98,E2 -12625.98} C_VEL
LIN {X 0,Y 368.916,Z 374.531,A -85,B 0,C 180,E1 -12629.69,E2 -12629.69} C_VEL
LIN {X 0,Y 368.9,Z 374.531,A -85,B 0,C 180,E1 -12633.044,E2 -12633.044} C_VEL
LIN {X 0,Y 368.92,Z 374.532,A -85,B 0,C 180,E1 -12636.197,E2 -12636.197} C_VEL
LIN {X 0,Y 368.907,Z 374.53,A -85,B 0,C 180,E1 -12638.953,E2 -12638.953} C_VEL
LIN {X 0,Y 368.89,Z 374.536,A -85,B 0,C 180,E1 -12642.011,E2 -12642.011} C_VEL
LIN {X 0,Y 368.93,Z 374.529,A -85,B 0,C 180,E1 -12645.183,E2 -12645.183} C_VEL
LIN {X 0,Y 368.885,Z 374.535,A -85,B 0,C 180,E1 -12648.178,E2 -12648.178} C_VEL
LIN {X 0,Y 368.931,Z 374.528,A -85,B 0,C 180,E1 -12651.749,E2 -12651.749} C_VEL
LIN {X 0,Y 368.952,Z 374.55,A -85,B 0,C 180,E1 -12652.443,E2 -12652.443} C_VEL
LIN {X 0,Y 371.394,Z 386.34,A -85,B 0,C 180,E1 -12656.37,E2 -12656.37} C_VEL
LIN {X 0,Y 373.473,Z 396.063,A -85,B 0,C 180,E1 -12659.464,E2 -12659.464} C_VEL
LIN {X 0,Y 373.498,Z 400.267,A -85,B 0,C 180,E1 -12660.71,E2 -12660.71} C_VEL
LIN {X 0,Y 371.858,Z 412.642,A -85,B 0,C 180,E1 -12664.234,E2 -12664.234} C_VEL
LIN {X 0,Y 370.284,Z 426.577,A -85,B 0,C 180,E1 -12668.155,E2 -12668.155} C_VEL
LIN {X 0,Y 369.077,Z 441.345,A -85,B 0,C 180,E1 -12672.261,E2 -12672.261} C_VEL
LIN {X 0,Y 369.007,Z 442.073,A -85,B 0,C 180,E1 -12672.437,E2 -12672.437} C_VEL
LIN {X 0,Y 370.001,Z 455.687,A -85,B 0,C 180,E1 -12672.931,E2 -12672.931} C_VEL
LIN {X 0,Y 370.907,Z 467.458,A -85,B 0,C 180,E1 -12673.558,E2 -12673.558} C_VEL
LIN {X 0,Y 371.062,Z 472.953,A -85,B 0,C 180,E1 -12673.919,E2 -12673.919} C_VEL
LIN {X 0,Y 370.362,Z 485.059,A -85,B 0,C 180,E1 -12674.875,E2 -12674.875} C_VEL
LIN {X 0,Y 369.765,Z 494.953,A -85,B 0,C 180,E1 -12675.866,E2 -12675.866} C_VEL
LIN {X 0,Y 369.144,Z 504.678,A -85,B 0,C 180,E1 -12677.073,E2 -12677.073} C_VEL
LIN {X 0,Y 368.598,Z 513.668,A -85,B 0,C 180,E1 -12678.451,E2 -12678.451} C_VEL
LIN {X 0,Y 368.163,Z 521.023,A -85,B 0,C 180,E1 -12679.83,E2 -12679.83} C_VEL
LIN {X 0,Y 367.941,Z 528.174,A -85,B 0,C 180,E1 -12681.487,E2 -12681.487} C_VEL
LIN {X 0,Y 367.838,Z 534.572,A -85,B 0,C 180,E1 -12683.417,E2 -12683.417} C_VEL
LIN {X 0,Y 367.773,Z 538.66,A -85,B 0,C 180,E1 -12685.067,E2 -12685.067} C_VEL
LIN {X 0,Y 367.914,Z 541.608,A -85,B 0,C 180,E1 -12686.715,E2 -12686.715} C_VEL
LIN {X 0,Y 367.984,Z 542.95,A -85,B 0,C 180,E1 -12687.811,E2 -12687.811} C_VEL
LIN {X 0,Y 367.876,Z 543.831,A -85,B 0,C 180,E1 -12688.905,E2 -12688.905} C_VEL
LIN {X 0,Y 367.842,Z 544.297,A -85,B 0,C 180,E1 -12690,E2 -12690} C_VEL
LIN {X 0,Y 367.876,Z 544.292,A -85,B 0,C 180,E1 -12691.095,E2 -12691.095} C_VEL
LIN {X 0,Y 367.908,Z 543.864,A -85,B 0,C 180,E1 -12692.19,E2 -12692.19} C_VEL
LIN {X 0,Y 367.836,Z 543.011,A -85,B 0,C 180,E1 -12693.286,E2 -12693.286} C_VEL
LIN {X 0,Y 367.688,Z 541.678,A -85,B 0,C 180,E1 -12694.385,E2 -12694.385} C_VEL
LIN {X 0,Y 367.716,Z 538.204,A -85,B 0,C 180,E1 -12696.354,E2 -12696.354} C_VEL
LIN {X 0,Y 367.803,Z 533.469,A -85,B 0,C 180,E1 -12698.24,E2 -12698.24} C_VEL
LIN {X 0,Y 368.144,Z 526.966,A -85,B 0,C 180,E1 -12700.171,E2 -12700.171} C_VEL
LIN {X 0,Y 368.799,Z 519.938,A -85,B 0,C 180,E1 -12701.821,E2 -12701.821} C_VEL
LIN {X 0,Y 369.574,Z 511.143,A -85,B 0,C 180,E1 -12703.471,E2 -12703.471} C_VEL
LIN {X 0,Y 370.702,Z 501.219,A -85,B 0,C 180,E1 -12704.97,E2 -12704.97} C_VEL
LIN {X 0,Y 371.879,Z 489.9,A -85,B 0,C 180,E1 -12706.327,E2 -12706.327} C_VEL
LIN {X 0,Y 373.149,Z 478.541,A -85,B 0,C 180,E1 -12707.397,E2 -12707.397} C_VEL
LIN {X 0,Y 373.501,Z 470.678,A -85,B 0,C 180,E1 -12708.026,E2 -12708.026} C_VEL
LIN {X 0,Y 373.097,Z 457.942,A -85,B 0,C 180,E1 -12708.89,E2 -12708.89} C_VEL
LIN {X 0,Y 371.564,Z 446.521,A -85,B 0,C 180,E1 -12709.557,E2 -12709.557} C_VEL
LIN {X 0,Y 370.249,Z 440.007,A -85,B 0,C 180,E1 -12709.907,E2 -12709.907} C_VEL
LIN {X 0,Y 371.773,Z 428.342,A -85,B 0,C 180,E1 -12713.39,E2 -12713.39} C_VEL
LIN {X 0,Y 374.094,Z 415.938,A -85,B 0,C 180,E1 -12717.405,E2 -12717.405} C_VEL
LIN {X 0,Y 376.107,Z 407.814,A -85,B 0,C 180,E1 -12720.3,E2 -12720.3} C_VEL
LIN {X 0,Y 376.021,Z 404.911,A -85,B 0,C 180,E1 -12721.556,E2 -12721.556} C_VEL
LIN {X 0,Y 375.007,Z 399.256,A -85,B 0,C 180,E1 -12724.452,E2 -12724.452} C_VEL
LIN {X 0,Y 374.047,Z 395.331,A -85,B 0,C 180,E1 -12726.96,E2 -12726.96} C_VEL
LIN {X 0,Y 373.274,Z 391.829,A -85,B 0,C 180,E1 -12729.803,E2 -12729.803} C_VEL
LIN {X 0,Y 372.64,Z 389.308,A -85,B 0,C 180,E1 -12732.763,E2 -12732.763} C_VEL
LIN {X 0,Y 372.236,Z 387.892,A -85,B 0,C 180,E1 -12735.845,E2 -12735.845} C_VEL
LIN {X 0,Y 372.037,Z 387.575,A -85,B 0,C 180,E1 -12738.611,E2 -12738.611} C_VEL
LIN {X 0,Y 372.031,Z 388.078,A -85,B 0,C 180,E1 -12741.435,E2 -12741.435} C_VEL
LIN {X 0,Y 372.13,Z 389.36,A -85,B 0,C 180,E1 -12744.301,E2 -12744.301} C_VEL
LIN {X 0,Y 372.301,Z 391.051,A -85,B 0,C 180,E1 -12746.808,E2 -12746.808} C_VEL
LIN {X 0,Y 372.2,Z 393.28,A -85,B 0,C 180,E1 -12749.348,E2 -12749.348} C_VEL
LIN {X 0,Y 371.705,Z 395.959,A -85,B 0,C 180,E1 -12751.791,E2 -12751.791} C_VEL
LIN {X 0,Y 370.938,Z 400.358,A -85,B 0,C 180,E1 -12755.366,E2 -12755.366} C_VEL
LIN {X 0,Y 370.286,Z 405.095,A -85,B 0,C 180,E1 -12758.862,E2 -12758.862} C_VEL
LIN {X 0,Y 369.778,Z 410.101,A -85,B 0,C 180,E1 -12762.296,E2 -12762.296} C_VEL
LIN {X 0,Y 369.347,Z 415.155,A -85,B 0,C 180,E1 -12765.573,E2 -12765.573} C_VEL
LIN {X 0,Y 372.269,Z 425.832,A -85,B 0,C 180,E1 -12766.621,E2 -12766.621} C_VEL
LIN {X 0,Y 373.902,Z 435.616,A -85,B 0,C 180,E1 -12767.696,E2 -12767.696} C_VEL
LIN {X 0,Y 372.865,Z 445.532,A -85,B 0,C 180,E1 -12768.844,E2 -12768.844} C_VEL
LIN {X 0,Y 371.917,Z 453.249,A -85,B 0,C 180,E1 -12769.985,E2 -12769.985} C_VEL
LIN {X 0,Y 370.97,Z 460.148,A -85,B 0,C 180,E1 -12771.283,E2 -12771.283} C_VEL
LIN {X 0,Y 370.315,Z 464.7,A -85,B 0,C 180,E1 -12772.366,E2 -12772.366} C_VEL
LIN {X 0,Y 369.531,Z 469.932,A -85,B 0,C 180,E1 -12773.996,E2 -12773.996} C_VEL
LIN {X 0,Y 368.804,Z 473.463,A -85,B 0,C 180,E1 -12775.628,E2 -12775.628} C_VEL
LIN {X 0,Y 368.402,Z 474.941,A -85,B 0,C 180,E1 -12776.719,E2 -12776.719} C_VEL
LIN {X 0,Y 368.135,Z 475.746,A -85,B 0,C 180,E1 -12777.812,E2 -12777.812} C_VEL
LIN {X 0,Y 367.979,Z 475.894,A -85,B 0,C 180,E1 -12778.906,E2 -12778.906} C_VEL
LIN {X 0,Y 367.91,Z 475.384,A -85,B 0,C 180,E1 -12780,E2 -12780} C_VEL
LIN {X 0,Y 367.928,Z 474.213,A -85,B 0,C 180,E1 -12781.095,E2 -12781.095} C_VEL
LIN {X 0,Y 368.058,Z 471.168,A -85,B 0,C 180,E1 -12782.736,E2 -12782.736} C_VEL
LIN {X 0,Y 368.358,Z 466.442,A -85,B 0,C 180,E1 -12784.377,E2 -12784.377} C_VEL
LIN {X 0,Y 368.581,Z 461.04,A -85,B 0,C 180,E1 -12785.745,E2 -12785.745} C_VEL
LIN {X 0,Y 368.85,Z 454.002,A -85,B 0,C 180,E1 -12787.114,E2 -12787.114} C_VEL
LIN {X 0,Y 369.042,Z 445.856,A -85,B 0,C 180,E1 -12788.349,E2 -12788.349} C_VEL
LIN {X 0,Y 369.539,Z 436.583,A -85,B 0,C 180,E1 -12789.441,E2 -12789.441} C_VEL
LIN {X 0,Y 369.944,Z 427.682,A -85,B 0,C 180,E1 -12790.259,E2 -12790.259} C_VEL
LIN {X 0,Y 368.77,Z 417.867,A -85,B 0,C 180,E1 -12790.987,E2 -12790.987} C_VEL
LIN {X 0,Y 367.96,Z 410.376,A -85,B 0,C 180,E1 -12791.43,E2 -12791.43} C_VEL
LIN {X 0,Y 368.081,Z 403.781,A -85,B 0,C 180,E1 -12794.938,E2 -12794.938} C_VEL
LIN {X 0,Y 368.257,Z 398.529,A -85,B 0,C 180,E1 -12797.78,E2 -12797.78} C_VEL
LIN {X 0,Y 368.5,Z 392.238,A -85,B 0,C 180,E1 -12801.246,E2 -12801.246} C_VEL
LIN {X 0,Y 368.75,Z 385.907,A -85,B 0,C 180,E1 -12804.79,E2 -12804.79} C_VEL
LIN {X 0,Y 369.144,Z 378.776,A -85,B 0,C 180,E1 -12808.862,E2 -12808.862} C_VEL
LIN {X 0,Y 369.108,Z 374.509,A -85,B 0,C 180,E1 -12811.378,E2 -12811.378} C_VEL
LIN {X 0,Y 368.932,Z 374.531,A -85,B 0,C 180,E1 -12815.002,E2 -12815.002} C_VEL
LIN {X 0,Y 368.914,Z 374.533,A -85,B 0,C 180,E1 -12818.641,E2 -12818.641} C_VEL
LIN {X 0,Y 368.884,Z 374.533,A -85,B 0,C 180,E1 -12822.009,E2 -12822.009} C_VEL
LIN {X 0,Y 368.91,Z 374.532,A -85,B 0,C 180,E1 -12825.18,E2 -12825.18} C_VEL
LIN {X 0,Y 368.886,Z 374.534,A -85,B 0,C 180,E1 -12828.178,E2 -12828.178} C_VEL
LIN {X 0,Y 368.911,Z 374.53,A -85,B 0,C 180,E1 -12831.36,E2 -12831.36} C_VEL
LIN {X 0,Y 368.939,Z 374.527,A -85,B 0,C 180,E1 -12835.147,E2 -12835.147} C_VEL
LIN {X 0,Y 368.932,Z 374.529,A -85,B 0,C 180,E1 -12839.047,E2 -12839.047} C_VEL
LIN {X 0,Y 368.966,Z 374.526,A -85,B 0,C 180,E1 -12842.797,E2 -12842.797} C_VEL
LIN {X 0,Y 368.948,Z 374.528,A -85,B 0,C 180,E1 -12846.113,E2 -12846.113} C_VEL
LIN {X 0,Y 368.94,Z 374.529,A -85,B 0,C 180,E1 -12849.947,E2 -12849.947} C_VEL
LIN {X 0,Y 368.979,Z 374.521,A -85,B 0,C 180,E1 -12853.399,E2 -12853.399} C_VEL
LIN {X 0,Y 369.061,Z 374.511,A -85,B 0,C 180,E1 -12856.79,E2 -12856.79} C_VEL
LIN {X 0,Y 369.071,Z 374.514,A -85,B 0,C 180,E1 -12860.132,E2 -12860.132} C_VEL
LIN {X 0,Y 369.203,Z 374.494,A -85,B 0,C 180,E1 -12863.442,E2 -12863.442} C_VEL
LIN {X 0,Y 369.32,Z 374.482,A -85,B 0,C 180,E1 -12867.819,E2 -12867.819} C_VEL
LIN {X 0,Y 369.46,Z 374.466,A -85,B 0,C 180,E1 -12870,E2 -12870} C_VEL
LIN {X 0,Y 369.323,Z 374.482,A -85,B 0,C 180,E1 -12872.181,E2 -12872.181} C_VEL
LIN {X 0,Y 369.202,Z 374.494,A -85,B 0,C 180,E1 -12876.558,E2 -12876.558} C_VEL
LIN {X 0,Y 369.126,Z 374.502,A -85,B 0,C 180,E1 -12878.761,E2 -12878.761} C_VEL
LIN {X 0,Y 369.009,Z 374.521,A -85,B 0,C 180,E1 -12882.093,E2 -12882.093} C_VEL
LIN {X 0,Y 369.001,Z 374.522,A -85,B 0,C 180,E1 -12885.465,E2 -12885.465} C_VEL
LIN {X 0,Y 368.993,Z 374.519,A -85,B 0,C 180,E1 -12888.892,E2 -12888.892} C_VEL
LIN {X 0,Y 368.94,Z 374.526,A -85,B 0,C 180,E1 -12892.395,E2 -12892.395} C_VEL
LIN {X 0,Y 369.003,Z 374.521,A -85,B 0,C 180,E1 -12895.98,E2 -12895.98} C_VEL
LIN {X 0,Y 368.917,Z 374.533,A -85,B 0,C 180,E1 -12899.69,E2 -12899.69} C_VEL
LIN {X 0,Y 368.899,Z 374.533,A -85,B 0,C 180,E1 -12903.043,E2 -12903.043} C_VEL
LIN {X 0,Y 368.92,Z 374.529,A -85,B 0,C 180,E1 -12906.197,E2 -12906.197} C_VEL
LIN {X 0,Y 368.893,Z 374.532,A -85,B 0,C 180,E1 -12909.179,E2 -12909.179} C_VEL
LIN {X 0,Y 368.884,Z 374.533,A -85,B 0,C 180,E1 -12912.009,E2 -12912.009} C_VEL
LIN {X 0,Y 368.868,Z 374.535,A -85,B 0,C 180,E1 -12913.925,E2 -12913.925} C_VEL
LIN {X 0,Y 368.188,Z 374.623,A -85,B 0,C 180,E1 -12914.837,E2 -12914.837} C_VEL
LIN {X 0,Y 365.339,Z 374.975,A -85,B 0,C 180,E1 -12916.319,E2 -12916.319} C_VEL
LIN {X 0,Y 362.937,Z 375.277,A -85,B 0,C 180,E1 -12917.518,E2 -12917.518} C_VEL
LIN {X 0,Y 361.91,Z 375.403,A -85,B 0,C 180,E1 -12918.446,E2 -12918.446} C_VEL
LIN {X 0,Y 361.828,Z 375.414,A -85,B 0,C 180,E1 -12918.76,E2 -12918.76} C_VEL
LIN {X 0,Y 361.87,Z 375.408,A -85,B 0,C 180,E1 -12921.575,E2 -12921.575} C_VEL
LIN {X 0,Y 361.876,Z 375.408,A -85,B 0,C 180,E1 -12924.655,E2 -12924.655} C_VEL
LIN {X 0,Y 361.839,Z 375.411,A -85,B 0,C 180,E1 -12928.37,E2 -12928.37} C_VEL
LIN {X 0,Y 361.902,Z 375.407,A -85,B 0,C 180,E1 -12930.955,E2 -12930.955} C_VEL
LIN {X 0,Y 361.957,Z 375.396,A -85,B 0,C 180,E1 -12933.475,E2 -12933.475} C_VEL
LIN {X 0,Y 361.892,Z 375.407,A -85,B 0,C 180,E1 -12937.145,E2 -12937.145} C_VEL
LIN {X 0,Y 361.909,Z 375.406,A -85,B 0,C 180,E1 -12940.723,E2 -12940.723} C_VEL
LIN {X 0,Y 361.935,Z 375.401,A -85,B 0,C 180,E1 -12943.066,E2 -12943.066} C_VEL
LIN {X 0,Y 362.003,Z 375.394,A -85,B 0,C 180,E1 -12946.528,E2 -12946.528} C_VEL
LIN {X 0,Y 362.038,Z 375.386,A -85,B 0,C 180,E1 -12949.938,E2 -12949.938} C_VEL
LIN {X 0,Y 362.154,Z 375.374,A -85,B 0,C 180,E1 -12952.193,E2 -12952.193} C_VEL
LIN {X 0,Y 362.12,Z 375.379,A -85,B 0,C 180,E1 -12954.431,E2 -12954.431} C_VEL
LIN {X 0,Y 362.283,Z 375.355,A -85,B 0,C 180,E1 -12957.776,E2 -12957.776} C_VEL
LIN {X 0,Y 362.43,Z 375.339,A -85,B 0,C 180,E1 -12960,E2 -12960} C_VEL
LIN {X 0,Y 362.285,Z 375.359,A -85,B 0,C 180,E1 -12962.223,E2 -12962.223} C_VEL
LIN {X 0,Y 362.174,Z 375.371,A -85,B 0,C 180,E1 -12966.686,E2 -12966.686} C_VEL
LIN {X 0,Y 362.076,Z 375.382,A -85,B 0,C 180,E1 -12968.933,E2 -12968.933} C_VEL
LIN {X 0,Y 361.963,Z 375.399,A -85,B 0,C 180,E1 -12972.332,E2 -12972.332} C_VEL
LIN {X 0,Y 361.964,Z 375.398,A -85,B 0,C 180,E1 -12974.62,E2 -12974.62} C_VEL
LIN {X 0,Y 361.961,Z 375.4,A -85,B 0,C 180,E1 -12978.099,E2 -12978.099} C_VEL
LIN {X 0,Y 361.894,Z 375.405,A -85,B 0,C 180,E1 -12981.653,E2 -12981.653} C_VEL
LIN {X 0,Y 361.93,Z 375.4,A -85,B 0,C 180,E1 -12985.29,E2 -12985.29} C_VEL
LIN {X 0,Y 361.91,Z 375.405,A -85,B 0,C 180,E1 -12987.779,E2 -12987.779} C_VEL
LIN {X 0,Y 361.839,Z 375.413,A -85,B 0,C 180,E1 -12991.629,E2 -12991.629} C_VEL
LIN {X 0,Y 361.876,Z 375.407,A -85,B 0,C 180,E1 -12995.345,E2 -12995.345} C_VEL
LIN {X 0,Y 361.874,Z 375.406,A -85,B 0,C 180,E1 -12999.027,E2 -12999.027} C_VEL
LIN {X 0,Y 361.84,Z 375.41,A -85,B 0,C 180,E1 -13002.828,E2 -13002.828} C_VEL
LIN {X 0,Y 361.854,Z 375.413,A -85,B 0,C 180,E1 -13005.941,E2 -13005.941} C_VEL
LIN {X 0,Y 361.837,Z 375.413,A -85,B 0,C 180,E1 -13009.245,E2 -13009.245} C_VEL
LIN {X 0,Y 361.919,Z 375.503,A -85,B 0,C 180,E1 -13012.122,E2 -13012.122} C_VEL
LIN {X 0,Y 364.281,Z 386.996,A -85,B 0,C 180,E1 -13016.057,E2 -13016.057} C_VEL
LIN {X 0,Y 366.586,Z 397.989,A -85,B 0,C 180,E1 -13019.623,E2 -13019.623} C_VEL
LIN {X 0,Y 366.448,Z 401.646,A -85,B 0,C 180,E1 -13020.721,E2 -13020.721} C_VEL
LIN {X 0,Y 364.758,Z 413.949,A -85,B 0,C 180,E1 -13024.309,E2 -13024.309} C_VEL
LIN {X 0,Y 363.104,Z 428.239,A -85,B 0,C 180,E1 -13028.423,E2 -13028.423} C_VEL
LIN {X 0,Y 362.047,Z 440.871,A -85,B 0,C 180,E1 -13032.024,E2 -13032.024} C_VEL
LIN {X 0,Y 361.957,Z 441.677,A -85,B 0,C 180,E1 -13032.252,E2 -13032.252} C_VEL
LIN {X 0,Y 362.986,Z 456.302,A -85,B 0,C 180,E1 -13032.812,E2 -13032.812} C_VEL
LIN {X 0,Y 363.91,Z 468.775,A -85,B 0,C 180,E1 -13033.522,E2 -13033.522} C_VEL
LIN {X 0,Y 363.96,Z 474.021,A -85,B 0,C 180,E1 -13033.884,E2 -13033.884} C_VEL
LIN {X 0,Y 363.268,Z 485.798,A -85,B 0,C 180,E1 -13034.86,E2 -13034.86} C_VEL
LIN {X 0,Y 362.513,Z 496.581,A -85,B 0,C 180,E1 -13036.01,E2 -13036.01} C_VEL
LIN {X 0,Y 362.027,Z 504.919,A -85,B 0,C 180,E1 -13037.1,E2 -13037.1} C_VEL
LIN {X 0,Y 361.478,Z 513.764,A -85,B 0,C 180,E1 -13038.505,E2 -13038.505} C_VEL
LIN {X 0,Y 361.073,Z 521,A -85,B 0,C 180,E1 -13039.911,E2 -13039.911} C_VEL
LIN {X 0,Y 360.862,Z 527.991,A -85,B 0,C 180,E1 -13041.601,E2 -13041.601} C_VEL
LIN {X 0,Y 360.792,Z 533.914,A -85,B 0,C 180,E1 -13043.439,E2 -13043.439} C_VEL
LIN {X 0,Y 360.719,Z 537.66,A -85,B 0,C 180,E1 -13044.97,E2 -13044.97} C_VEL
LIN {X 0,Y 360.85,Z 540.69,A -85,B 0,C 180,E1 -13046.65,E2 -13046.65} C_VEL
LIN {X 0,Y 360.937,Z 542.109,A -85,B 0,C 180,E1 -13047.768,E2 -13047.768} C_VEL
LIN {X 0,Y 360.83,Z 543.024,A -85,B 0,C 180,E1 -13048.884,E2 -13048.884} C_VEL
LIN {X 0,Y 360.794,Z 543.527,A -85,B 0,C 180,E1 -13050,E2 -13050} C_VEL
LIN {X 0,Y 360.829,Z 543.588,A -85,B 0,C 180,E1 -13051.116,E2 -13051.116} C_VEL
LIN {X 0,Y 360.833,Z 543.186,A -85,B 0,C 180,E1 -13052.233,E2 -13052.233} C_VEL
LIN {X 0,Y 360.753,Z 542.366,A -85,B 0,C 180,E1 -13053.351,E2 -13053.351} C_VEL
LIN {X 0,Y 360.609,Z 541.099,A -85,B 0,C 180,E1 -13054.471,E2 -13054.471} C_VEL
LIN {X 0,Y 360.619,Z 538.022,A -85,B 0,C 180,E1 -13056.318,E2 -13056.318} C_VEL
LIN {X 0,Y 360.744,Z 533.049,A -85,B 0,C 180,E1 -13058.402,E2 -13058.402} C_VEL
LIN {X 0,Y 361.085,Z 526.66,A -85,B 0,C 180,E1 -13060.372,E2 -13060.372} C_VEL
LIN {X 0,Y 361.81,Z 519.737,A -85,B 0,C 180,E1 -13062.053,E2 -13062.053} C_VEL
LIN {X 0,Y 362.643,Z 511.179,A -85,B 0,C 180,E1 -13063.725,E2 -13063.725} C_VEL
LIN {X 0,Y 363.715,Z 502.342,A -85,B 0,C 180,E1 -13065.121,E2 -13065.121} C_VEL
LIN {X 0,Y 364.977,Z 491.591,A -85,B 0,C 180,E1 -13066.501,E2 -13066.501} C_VEL
LIN {X 0,Y 366.436,Z 479.367,A -85,B 0,C 180,E1 -13067.727,E2 -13067.727} C_VEL
LIN {X 0,Y 366.851,Z 471.398,A -85,B 0,C 180,E1 -13068.396,E2 -13068.396} C_VEL
LIN {X 0,Y 366.644,Z 459.879,A -85,B 0,C 180,E1 -13069.236,E2 -13069.236} C_VEL
LIN {X 0,Y 365.308,Z 448.755,A -85,B 0,C 180,E1 -13069.944,E2 -13069.944} C_VEL
LIN {X 0,Y 363.476,Z 439.594,A -85,B 0,C 180,E1 -13070.478,E2 -13070.478} C_VEL
LIN {X 0,Y 365.013,Z 428.691,A -85,B 0,C 180,E1 -13073.85,E2 -13073.85} C_VEL
LIN {X 0,Y 367.116,Z 418.19,A -85,B 0,C 180,E1 -13077.352,E2 -13077.352} C_VEL
LIN {X 0,Y 369.249,Z 410.117,A -85,B 0,C 180,E1 -13080.29,E2 -13080.29} C_VEL
LIN {X 0,Y 369.385,Z 408.187,A -85,B 0,C 180,E1 -13081.109,E2 -13081.109} C_VEL
LIN {X 0,Y 368.661,Z 403.252,A -85,B 0,C 180,E1 -13083.563,E2 -13083.563} C_VEL
LIN {X 0,Y 367.565,Z 398.357,A -85,B 0,C 180,E1 -13086.577,E2 -13086.577} C_VEL
LIN {X 0,Y 366.624,Z 394.244,A -85,B 0,C 180,E1 -13089.934,E2 -13089.934} C_VEL
LIN {X 0,Y 366.125,Z 392.285,A -85,B 0,C 180,E1 -13092.21,E2 -13092.21} C_VEL
LIN {X 0,Y 365.651,Z 390.61,A -85,B 0,C 180,E1 -13095.33,E2 -13095.33} C_VEL
LIN {X 0,Y 365.449,Z 390.097,A -85,B 0,C 180,E1 -13097.694,E2 -13097.694} C_VEL
LIN {X 0,Y 365.379,Z 390.268,A -85,B 0,C 180,E1 -13100.599,E2 -13100.599} C_VEL
LIN {X 0,Y 365.388,Z 391.456,A -85,B 0,C 180,E1 -13103.886,E2 -13103.886} C_VEL
LIN {X 0,Y 365.517,Z 392.724,A -85,B 0,C 180,E1 -13106.11,E2 -13106.11} C_VEL
LIN {X 0,Y 365.449,Z 394.823,A -85,B 0,C 180,E1 -13108.719,E2 -13108.719} C_VEL
LIN {X 0,Y 365.004,Z 397.318,A -85,B 0,C 180,E1 -13111.225,E2 -13111.225} C_VEL
LIN {X 0,Y 364.143,Z 401.569,A -85,B 0,C 180,E1 -13114.874,E2 -13114.874} C_VEL
LIN {X 0,Y 363.448,Z 406.23,A -85,B 0,C 180,E1 -13118.444,E2 -13118.444} C_VEL
LIN {X 0,Y 362.9,Z 411.169,A -85,B 0,C 180,E1 -13121.949,E2 -13121.949} C_VEL
LIN {X 0,Y 362.476,Z 415.818,A -85,B 0,C 180,E1 -13125.005,E2 -13125.005} C_VEL
LIN {X 0,Y 365.59,Z 426.653,A -85,B 0,C 180,E1 -13126.128,E2 -13126.128} C_VEL
LIN {X 0,Y 367.209,Z 435.791,A -85,B 0,C 180,E1 -13127.174,E2 -13127.174} C_VEL
LIN {X 0,Y 367.18,Z 438.95,A -85,B 0,C 180,E1 -13127.537,E2 -13127.537} C_VEL
LIN {X 0,Y 366.091,Z 448.054,A -85,B 0,C 180,E1 -13128.687,E2 -13128.687} C_VEL
LIN {X 0,Y 364.919,Z 456.331,A -85,B 0,C 180,E1 -13130.018,E2 -13130.018} C_VEL
LIN {X 0,Y 363.972,Z 462.929,A -85,B 0,C 180,E1 -13131.394,E2 -13131.394} C_VEL
LIN {X 0,Y 363.18,Z 468.011,A -85,B 0,C 180,E1 -13132.774,E2 -13132.774} C_VEL
LIN {X 0,Y 362.269,Z 472.445,A -85,B 0,C 180,E1 -13134.434,E2 -13134.434} C_VEL
LIN {X 0,Y 361.799,Z 474.488,A -85,B 0,C 180,E1 -13135.544,E2 -13135.544} C_VEL
LIN {X 0,Y 361.376,Z 475.872,A -85,B 0,C 180,E1 -13136.655,E2 -13136.655} C_VEL
LIN {X 0,Y 361.091,Z 476.584,A -85,B 0,C 180,E1 -13137.769,E2 -13137.769} C_VEL
LIN {X 0,Y 360.928,Z 476.634,A -85,B 0,C 180,E1 -13138.884,E2 -13138.884} C_VEL
LIN {X 0,Y 360.858,Z 476.025,A -85,B 0,C 180,E1 -13140,E2 -13140} C_VEL
LIN {X 0,Y 360.879,Z 474.755,A -85,B 0,C 180,E1 -13141.116,E2 -13141.116} C_VEL
LIN {X 0,Y 360.986,Z 471.573,A -85,B 0,C 180,E1 -13142.79,E2 -13142.79} C_VEL
LIN {X 0,Y 361.285,Z 466.72,A -85,B 0,C 180,E1 -13144.463,E2 -13144.463} C_VEL
LIN {X 0,Y 361.514,Z 461.173,A -85,B 0,C 180,E1 -13145.858,E2 -13145.858} C_VEL
LIN {X 0,Y 361.795,Z 454.215,A -85,B 0,C 180,E1 -13147.211,E2 -13147.211} C_VEL
LIN {X 0,Y 361.99,Z 445.946,A -85,B 0,C 180,E1 -13148.471,E2 -13148.471} C_VEL
LIN {X 0,Y 362.51,Z 436.124,A -85,B 0,C 180,E1 -13149.626,E2 -13149.626} C_VEL
LIN {X 0,Y 362.851,Z 426.978,A -85,B 0,C 180,E1 -13150.462,E2 -13150.462} C_VEL
LIN {X 0,Y 361.55,Z 416.755,A -85,B 0,C 180,E1 -13151.209,E2 -13151.209} C_VEL
LIN {X 0,Y 360.875,Z 410.642,A -85,B 0,C 180,E1 -13151.586,E2 -13151.586} C_VEL
LIN {X 0,Y 360.99,Z 404.932,A -85,B 0,C 180,E1 -13154.661,E2 -13154.661} C_VEL
LIN {X 0,Y 361.184,Z 399.644,A -85,B 0,C 180,E1 -13157.549,E2 -13157.549} C_VEL
LIN {X 0,Y 361.41,Z 393.391,A -85,B 0,C 180,E1 -13161.026,E2 -13161.026} C_VEL
LIN {X 0,Y 361.692,Z 386.917,A -85,B 0,C 180,E1 -13164.694,E2 -13164.694} C_VEL
LIN {X 0,Y 362.05,Z 380.51,A -85,B 0,C 180,E1 -13168.398,E2 -13168.398} C_VEL
LIN {X 0,Y 362.2,Z 377.26,A -85,B 0,C 180,E1 -13170.298,E2 -13170.298} C_VEL
LIN {X 0,Y 362.056,Z 375.387,A -85,B 0,C 180,E1 -13171.472,E2 -13171.472} C_VEL
LIN {X 0,Y 361.871,Z 375.407,A -85,B 0,C 180,E1 -13175.637,E2 -13175.637} C_VEL
LIN {X 0,Y 361.874,Z 375.411,A -85,B 0,C 180,E1 -13179.027,E2 -13179.027} C_VEL
LIN {X 0,Y 361.839,Z 375.416,A -85,B 0,C 180,E1 -13182.829,E2 -13182.829} C_VEL
LIN {X 0,Y 361.832,Z 375.411,A -85,B 0,C 180,E1 -13185.945,E2 -13185.945} C_VEL
LIN {X 0,Y 361.839,Z 375.412,A -85,B 0,C 180,E1 -13189.245,E2 -13189.245} C_VEL
LIN {X 0,Y 361.866,Z 375.411,A -85,B 0,C 180,E1 -13192.777,E2 -13192.777} C_VEL
LIN {X 0,Y 361.857,Z 375.408,A -85,B 0,C 180,E1 -13195.72,E2 -13195.72} C_VEL
LIN {X 0,Y 361.876,Z 375.406,A -85,B 0,C 180,E1 -13199.672,E2 -13199.672} C_VEL
LIN {X 0,Y 361.957,Z 375.396,A -85,B 0,C 180,E1 -13203.475,E2 -13203.475} C_VEL
LIN {X 0,Y 361.893,Z 375.404,A -85,B 0,C 180,E1 -13207.145,E2 -13207.145} C_VEL
LIN {X 0,Y 361.924,Z 375.402,A -85,B 0,C 180,E1 -13210.724,E2 -13210.724} C_VEL
LIN {X 0,Y 361.949,Z 375.401,A -85,B 0,C 180,E1 -13214.226,E2 -13214.226} C_VEL
LIN {X 0,Y 362.002,Z 375.393,A -85,B 0,C 180,E1 -13216.528,E2 -13216.528} C_VEL
LIN {X 0,Y 362.035,Z 375.39,A -85,B 0,C 180,E1 -13219.938,E2 -13219.938} C_VEL
LIN {X 0,Y 362.165,Z 375.37,A -85,B 0,C 180,E1 -13223.314,E2 -13223.314} C_VEL
LIN {X 0,Y 362.284,Z 375.358,A -85,B 0,C 180,E1 -13227.776,E2 -13227.776} C_VEL
LIN {X 0,Y 362.43,Z 375.341,A -85,B 0,C 180,E1 -13230,E2 -13230} C_VEL
LIN {X 0,Y 362.287,Z 375.359,A -85,B 0,C 180,E1 -13232.223,E2 -13232.223} C_VEL
LIN {X 0,Y 362.164,Z 375.37,A -85,B 0,C 180,E1 -13236.686,E2 -13236.686} C_VEL
LIN {X 0,Y 362.037,Z 375.389,A -85,B 0,C 180,E1 -13240.062,E2 -13240.062} C_VEL
LIN {X 0,Y 362.001,Z 375.395,A -85,B 0,C 180,E1 -13243.899,E2 -13243.899} C_VEL
LIN {X 0,Y 361.971,Z 375.397,A -85,B 0,C 180,E1 -13247.939,E2 -13247.939} C_VEL
LIN {X 0,Y 361.902,Z 375.407,A -85,B 0,C 180,E1 -13251.652,E2 -13251.652} C_VEL
LIN {X 0,Y 361.931,Z 375.403,A -85,B 0,C 180,E1 -13255.29,E2 -13255.29} C_VEL
LIN {X 0,Y 361.911,Z 375.405,A -85,B 0,C 180,E1 -13257.779,E2 -13257.779} C_VEL
LIN {X 0,Y 361.84,Z 375.414,A -85,B 0,C 180,E1 -13261.629,E2 -13261.629} C_VEL
LIN {X 0,Y 361.877,Z 375.41,A -85,B 0,C 180,E1 -13265.345,E2 -13265.345} C_VEL
LIN {X 0,Y 361.873,Z 375.409,A -85,B 0,C 180,E1 -13269.027,E2 -13269.027} C_VEL
LIN {X 0,Y 361.838,Z 375.412,A -85,B 0,C 180,E1 -13272.829,E2 -13272.829} C_VEL
LIN {X 0,Y 361.82,Z 375.414,A -85,B 0,C 180,E1 -13275.946,E2 -13275.946} C_VEL
LIN {X 0,Y 361.828,Z 375.414,A -85,B 0,C 180,E1 -13278.76,E2 -13278.76} C_VEL
LIN {X 0,Y 361.164,Z 375.499,A -85,B 0,C 180,E1 -13279.689,E2 -13279.689} C_VEL
LIN {X 0,Y 358.314,Z 375.857,A -85,B 0,C 180,E1 -13281.199,E2 -13281.199} C_VEL
LIN {X 0,Y 355.905,Z 376.155,A -85,B 0,C 180,E1 -13282.422,E2 -13282.422} C_VEL
LIN {X 0,Y 354.879,Z 376.28,A -85,B 0,C 180,E1 -13283.367,E2 -13283.367} C_VEL
LIN {X 0,Y 354.8,Z 376.288,A -85,B 0,C 180,E1 -13283.688,E2 -13283.688} C_VEL
LIN {X 0,Y 354.816,Z 376.286,A -85,B 0,C 180,E1 -13286.316,E2 -13286.316} C_VEL
LIN {X 0,Y 354.856,Z 376.281,A -85,B 0,C 180,E1 -13290.321,E2 -13290.321} C_VEL
LIN {X 0,Y 354.901,Z 376.274,A -85,B 0,C 180,E1 -13294.173,E2 -13294.173} C_VEL
LIN {X 0,Y 354.837,Z 376.283,A -85,B 0,C 180,E1 -13297.894,E2 -13297.894} C_VEL
LIN {X 0,Y 354.924,Z 376.272,A -85,B 0,C 180,E1 -13301.891,E2 -13301.891} C_VEL
LIN {X 0,Y 354.945,Z 376.269,A -85,B 0,C 180,E1 -13305.981,E2 -13305.981} C_VEL
LIN {X 0,Y 354.985,Z 376.264,A -85,B 0,C 180,E1 -13309.736,E2 -13309.736} C_VEL
LIN {X 0,Y 355.117,Z 376.249,A -85,B 0,C 180,E1 -13312.037,E2 -13312.037} C_VEL
LIN {X 0,Y 355.094,Z 376.254,A -85,B 0,C 180,E1 -13314.321,E2 -13314.321} C_VEL
LIN {X 0,Y 355.246,Z 376.232,A -85,B 0,C 180,E1 -13317.732,E2 -13317.732} C_VEL
LIN {X 0,Y 355.4,Z 376.214,A -85,B 0,C 180,E1 -13320,E2 -13320} C_VEL
LIN {X 0,Y 355.248,Z 376.236,A -85,B 0,C 180,E1 -13322.268,E2 -13322.268} C_VEL
LIN {X 0,Y 355.14,Z 376.246,A -85,B 0,C 180,E1 -13326.819,E2 -13326.819} C_VEL
LIN {X 0,Y 355.017,Z 376.26,A -85,B 0,C 180,E1 -13329.112,E2 -13329.112} C_VEL
LIN {X 0,Y 354.923,Z 376.275,A -85,B 0,C 180,E1 -13332.581,E2 -13332.581} C_VEL
LIN {X 0,Y 354.891,Z 376.28,A -85,B 0,C 180,E1 -13336.096,E2 -13336.096} C_VEL
LIN {X 0,Y 354.908,Z 376.277,A -85,B 0,C 180,E1 -13338.472,E2 -13338.472} C_VEL
LIN {X 0,Y 354.836,Z 376.287,A -85,B 0,C 180,E1 -13342.106,E2 -13342.106} C_VEL
LIN {X 0,Y 354.901,Z 376.278,A -85,B 0,C 180,E1 -13345.827,E2 -13345.827} C_VEL
LIN {X 0,Y 354.819,Z 376.287,A -85,B 0,C 180,E1 -13349.682,E2 -13349.682} C_VEL
LIN {X 0,Y 354.807,Z 376.29,A -85,B 0,C 180,E1 -13353.702,E2 -13353.702} C_VEL
LIN {X 0,Y 354.8,Z 376.288,A -85,B 0,C 180,E1 -13356.459,E2 -13356.459} C_VEL
LIN {X 0,Y 354.825,Z 376.286,A -85,B 0,C 180,E1 -13359.424,E2 -13359.424} C_VEL
LIN {X 0,Y 354.792,Z 376.288,A -85,B 0,C 180,E1 -13362.868,E2 -13362.868} C_VEL
LIN {X 0,Y 354.797,Z 376.29,A -85,B 0,C 180,E1 -13366.108,E2 -13366.108} C_VEL
LIN {X 0,Y 354.789,Z 376.29,A -85,B 0,C 180,E1 -13369.179,E2 -13369.179} C_VEL
LIN {X 0,Y 354.838,Z 376.285,A -85,B 0,C 180,E1 -13371.761,E2 -13371.761} C_VEL
LIN {X 0,Y 357.173,Z 387.663,A -85,B 0,C 180,E1 -13375.733,E2 -13375.733} C_VEL
LIN {X 0,Y 359.525,Z 398.827,A -85,B 0,C 180,E1 -13379.453,E2 -13379.453} C_VEL
LIN {X 0,Y 359.526,Z 401.951,A -85,B 0,C 180,E1 -13380.423,E2 -13380.423} C_VEL
LIN {X 0,Y 357.771,Z 414.211,A -85,B 0,C 180,E1 -13384.083,E2 -13384.083} C_VEL
LIN {X 0,Y 356.142,Z 427.607,A -85,B 0,C 180,E1 -13388.046,E2 -13388.046} C_VEL
LIN {X 0,Y 354.928,Z 441.419,A -85,B 0,C 180,E1 -13392.087,E2 -13392.087} C_VEL
LIN {X 0,Y 355.824,Z 455.283,A -85,B 0,C 180,E1 -13392.623,E2 -13392.623} C_VEL
LIN {X 0,Y 356.774,Z 467.658,A -85,B 0,C 180,E1 -13393.33,E2 -13393.33} C_VEL
LIN {X 0,Y 356.938,Z 473.012,A -85,B 0,C 180,E1 -13393.705,E2 -13393.705} C_VEL
LIN {X 0,Y 356.245,Z 484.876,A -85,B 0,C 180,E1 -13394.701,E2 -13394.701} C_VEL
LIN {X 0,Y 355.637,Z 494.414,A -85,B 0,C 180,E1 -13395.712,E2 -13395.712} C_VEL
LIN {X 0,Y 355.068,Z 503.156,A -85,B 0,C 180,E1 -13396.843,E2 -13396.843} C_VEL
LIN {X 0,Y 354.482,Z 512.184,A -85,B 0,C 180,E1 -13398.275,E2 -13398.275} C_VEL
LIN {X 0,Y 353.981,Z 520.911,A -85,B 0,C 180,E1 -13399.996,E2 -13399.996} C_VEL
LIN {X 0,Y 353.798,Z 527.776,A -85,B 0,C 180,E1 -13401.72,E2 -13401.72} C_VEL
LIN {X 0,Y 353.743,Z 533.065,A -85,B 0,C 180,E1 -13403.404,E2 -13403.404} C_VEL
LIN {X 0,Y 353.667,Z 536.638,A -85,B 0,C 180,E1 -13404.87,E2 -13404.87} C_VEL
LIN {X 0,Y 353.787,Z 539.753,A -85,B 0,C 180,E1 -13406.584,E2 -13406.584} C_VEL
LIN {X 0,Y 353.89,Z 541.244,A -85,B 0,C 180,E1 -13407.724,E2 -13407.724} C_VEL
LIN {X 0,Y 353.786,Z 542.206,A -85,B 0,C 180,E1 -13408.862,E2 -13408.862} C_VEL
LIN {X 0,Y 353.747,Z 542.745,A -85,B 0,C 180,E1 -13410,E2 -13410} C_VEL
LIN {X 0,Y 353.783,Z 542.87,A -85,B 0,C 180,E1 -13411.138,E2 -13411.138} C_VEL
LIN {X 0,Y 353.759,Z 542.511,A -85,B 0,C 180,E1 -13412.277,E2 -13412.277} C_VEL
LIN {X 0,Y 353.657,Z 541.721,A -85,B 0,C 180,E1 -13413.418,E2 -13413.418} C_VEL
LIN {X 0,Y 353.532,Z 540.516,A -85,B 0,C 180,E1 -13414.561,E2 -13414.561} C_VEL
LIN {X 0,Y 353.523,Z 537.846,A -85,B 0,C 180,E1 -13416.281,E2 -13416.281} C_VEL
LIN {X 0,Y 353.616,Z 534.135,A -85,B 0,C 180,E1 -13417.997,E2 -13417.997} C_VEL
LIN {X 0,Y 353.859,Z 529.283,A -85,B 0,C 180,E1 -13419.719,E2 -13419.719} C_VEL
LIN {X 0,Y 354.377,Z 523.167,A -85,B 0,C 180,E1 -13421.439,E2 -13421.439} C_VEL
LIN {X 0,Y 355.251,Z 515.609,A -85,B 0,C 180,E1 -13423.15,E2 -13423.15} C_VEL
LIN {X 0,Y 356.212,Z 507.572,A -85,B 0,C 180,E1 -13424.633,E2 -13424.633} C_VEL
LIN {X 0,Y 357.651,Z 496.565,A -85,B 0,C 180,E1 -13426.261,E2 -13426.261} C_VEL
LIN {X 0,Y 359.052,Z 485.857,A -85,B 0,C 180,E1 -13427.515,E2 -13427.515} C_VEL
LIN {X 0,Y 360.205,Z 475.59,A -85,B 0,C 180,E1 -13428.485,E2 -13428.485} C_VEL
LIN {X 0,Y 360.27,Z 463.137,A -85,B 0,C 180,E1 -13429.495,E2 -13429.495} C_VEL
LIN {X 0,Y 359.242,Z 452.409,A -85,B 0,C 180,E1 -13430.25,E2 -13430.25} C_VEL
LIN {X 0,Y 356.947,Z 440.648,A -85,B 0,C 180,E1 -13430.996,E2 -13430.996} C_VEL
LIN {X 0,Y 356.703,Z 439.248,A -85,B 0,C 180,E1 -13431.074,E2 -13431.074} C_VEL
LIN {X 0,Y 358.293,Z 429.113,A -85,B 0,C 180,E1 -13434.326,E2 -13434.326} C_VEL
LIN {X 0,Y 360.549,Z 418.785,A -85,B 0,C 180,E1 -13437.893,E2 -13437.893} C_VEL
LIN {X 0,Y 362.363,Z 412.424,A -85,B 0,C 180,E1 -13440.283,E2 -13440.283} C_VEL
LIN {X 0,Y 362.564,Z 409.681,A -85,B 0,C 180,E1 -13441.471,E2 -13441.471} C_VEL
LIN {X 0,Y 361.735,Z 404.353,A -85,B 0,C 180,E1 -13444.294,E2 -13444.294} C_VEL
LIN {X 0,Y 360.764,Z 400.158,A -85,B 0,C 180,E1 -13447.15,E2 -13447.15} C_VEL
LIN {X 0,Y 359.947,Z 396.613,A -85,B 0,C 180,E1 -13450.116,E2 -13450.116} C_VEL
LIN {X 0,Y 359.544,Z 394.982,A -85,B 0,C 180,E1 -13452.031,E2 -13452.031} C_VEL
LIN {X 0,Y 359.052,Z 393.221,A -85,B 0,C 180,E1 -13455.198,E2 -13455.198} C_VEL
LIN {X 0,Y 358.766,Z 392.585,A -85,B 0,C 180,E1 -13458.108,E2 -13458.108} C_VEL
LIN {X 0,Y 358.681,Z 392.828,A -85,B 0,C 180,E1 -13461.17,E2 -13461.17} C_VEL
LIN {X 0,Y 358.688,Z 393.832,A -85,B 0,C 180,E1 -13463.998,E2 -13463.998} C_VEL
LIN {X 0,Y 358.745,Z 395.394,A -85,B 0,C 180,E1 -13466.733,E2 -13466.733} C_VEL
LIN {X 0,Y 358.537,Z 397.741,A -85,B 0,C 180,E1 -13469.597,E2 -13469.597} C_VEL
LIN {X 0,Y 357.981,Z 400.24,A -85,B 0,C 180,E1 -13472.062,E2 -13472.062} C_VEL
LIN {X 0,Y 357.12,Z 404.324,A -85,B 0,C 180,E1 -13475.589,E2 -13475.589} C_VEL
LIN {X 0,Y 356.391,Z 408.998,A -85,B 0,C 180,E1 -13479.209,E2 -13479.209} C_VEL
LIN {X 0,Y 356.039,Z 412.262,A -85,B 0,C 180,E1 -13481.589,E2 -13481.589} C_VEL
LIN {X 0,Y 355.573,Z 416.284,A -85,B 0,C 180,E1 -13484.356,E2 -13484.356} C_VEL
LIN {X 0,Y 358.715,Z 426.692,A -85,B 0,C 180,E1 -13485.503,E2 -13485.503} C_VEL
LIN {X 0,Y 360.484,Z 435.927,A -85,B 0,C 180,E1 -13486.614,E2 -13486.614} C_VEL
LIN {X 0,Y 360.697,Z 439.984,A -85,B 0,C 180,E1 -13487.111,E2 -13487.111} C_VEL
LIN {X 0,Y 359.595,Z 448.656,A -85,B 0,C 180,E1 -13488.229,E2 -13488.229} C_VEL
LIN {X 0,Y 358.372,Z 456.721,A -85,B 0,C 180,E1 -13489.549,E2 -13489.549} C_VEL
LIN {X 0,Y 357.267,Z 463.35,A -85,B 0,C 180,E1 -13490.946,E2 -13490.946} C_VEL
LIN {X 0,Y 356.525,Z 467.568,A -85,B 0,C 180,E1 -13492.069,E2 -13492.069} C_VEL
LIN {X 0,Y 355.632,Z 472.363,A -85,B 0,C 180,E1 -13493.76,E2 -13493.76} C_VEL
LIN {X 0,Y 354.797,Z 475.533,A -85,B 0,C 180,E1 -13495.456,E2 -13495.456} C_VEL
LIN {X 0,Y 354.35,Z 476.798,A -85,B 0,C 180,E1 -13496.589,E2 -13496.589} C_VEL
LIN {X 0,Y 354.048,Z 477.407,A -85,B 0,C 180,E1 -13497.725,E2 -13497.725} C_VEL
LIN {X 0,Y 353.879,Z 477.362,A -85,B 0,C 180,E1 -13498.862,E2 -13498.862} C_VEL
LIN {X 0,Y 353.807,Z 476.657,A -85,B 0,C 180,E1 -13500,E2 -13500} C_VEL
LIN {X 0,Y 353.827,Z 474.349,A -85,B 0,C 180,E1 -13501.707,E2 -13501.707} C_VEL
LIN {X 0,Y 354.007,Z 470.47,A -85,B 0,C 180,E1 -13503.415,E2 -13503.415} C_VEL
LIN {X 0,Y 354.368,Z 464.817,A -85,B 0,C 180,E1 -13505.12,E2 -13505.12} C_VEL
LIN {X 0,Y 354.58,Z 458.513,A -85,B 0,C 180,E1 -13506.544,E2 -13506.544} C_VEL
LIN {X 0,Y 354.849,Z 450.337,A -85,B 0,C 180,E1 -13507.969,E2 -13507.969} C_VEL
LIN {X 0,Y 355.231,Z 442.009,A -85,B 0,C 180,E1 -13509.107,E2 -13509.107} C_VEL
LIN {X 0,Y 355.652,Z 432.744,A -85,B 0,C 180,E1 -13510.101,E2 -13510.101} C_VEL
LIN {X 0,Y 355.652,Z 426.179,A -85,B 0,C 180,E1 -13510.676,E2 -13510.676} C_VEL
LIN {X 0,Y 354.316,Z 415.552,A -85,B 0,C 180,E1 -13511.441,E2 -13511.441} C_VEL
LIN {X 0,Y 353.795,Z 410.896,A -85,B 0,C 180,E1 -13511.748,E2 -13511.748} C_VEL
LIN {X 0,Y 353.936,Z 405.007,A -85,B 0,C 180,E1 -13514.96,E2 -13514.96} C_VEL
LIN {X 0,Y 354.136,Z 400.035,A -85,B 0,C 180,E1 -13517.714,E2 -13517.714} C_VEL
LIN {X 0,Y 354.357,Z 393.819,A -85,B 0,C 180,E1 -13521.226,E2 -13521.226} C_VEL
LIN {X 0,Y 354.641,Z 387.931,A -85,B 0,C 180,E1 -13524.593,E2 -13524.593} C_VEL
LIN {X 0,Y 354.998,Z 381.485,A -85,B 0,C 180,E1 -13528.368,E2 -13528.368} C_VEL
LIN {X 0,Y 355.183,Z 378.219,A -85,B 0,C 180,E1 -13530.303,E2 -13530.303} C_VEL
LIN {X 0,Y 354.982,Z 376.267,A -85,B 0,C 180,E1 -13531.644,E2 -13531.644} C_VEL
LIN {X 0,Y 354.825,Z 376.284,A -85,B 0,C 180,E1 -13535.699,E2 -13535.699} C_VEL
LIN {X 0,Y 354.827,Z 376.285,A -85,B 0,C 180,E1 -13539.424,E2 -13539.424} C_VEL
LIN {X 0,Y 354.791,Z 376.293,A -85,B 0,C 180,E1 -13542.867,E2 -13542.867} C_VEL
LIN {X 0,Y 354.779,Z 376.29,A -85,B 0,C 180,E1 -13546.105,E2 -13546.105} C_VEL
LIN {X 0,Y 354.791,Z 376.29,A -85,B 0,C 180,E1 -13549.179,E2 -13549.179} C_VEL
LIN {X 0,Y 354.81,Z 376.29,A -85,B 0,C 180,E1 -13552.403,E2 -13552.403} C_VEL
LIN {X 0,Y 354.815,Z 376.288,A -85,B 0,C 180,E1 -13554.941,E2 -13554.941} C_VEL
LIN {X 0,Y 354.796,Z 376.293,A -85,B 0,C 180,E1 -13558.405,E2 -13558.405} C_VEL
LIN {X 0,Y 354.849,Z 376.281,A -85,B 0,C 180,E1 -13561.619,E2 -13561.619} C_VEL
LIN {X 0,Y 354.902,Z 376.278,A -85,B 0,C 180,E1 -13564.173,E2 -13564.173} C_VEL
LIN {X 0,Y 354.838,Z 376.284,A -85,B 0,C 180,E1 -13567.894,E2 -13567.894} C_VEL
LIN {X 0,Y 354.926,Z 376.274,A -85,B 0,C 180,E1 -13571.891,E2 -13571.891} C_VEL
LIN {X 0,Y 354.946,Z 376.272,A -85,B 0,C 180,E1 -13575.981,E2 -13575.981} C_VEL
LIN {X 0,Y 354.981,Z 376.266,A -85,B 0,C 180,E1 -13579.736,E2 -13579.736} C_VEL
LIN {X 0,Y 355.128,Z 376.246,A -85,B 0,C 180,E1 -13583.18,E2 -13583.18} C_VEL
LIN {X 0,Y 355.247,Z 376.234,A -85,B 0,C 180,E1 -13587.732,E2 -13587.732} C_VEL
LIN {X 0,Y 355.4,Z 376.217,A -85,B 0,C 180,E1 -13590,E2 -13590} C_VEL
LIN {X 0,Y 355.249,Z 376.234,A -85,B 0,C 180,E1 -13592.268,E2 -13592.268} C_VEL
LIN {X 0,Y 355.129,Z 376.246,A -85,B 0,C 180,E1 -13596.819,E2 -13596.819} C_VEL
LIN {X 0,Y 354.983,Z 376.266,A -85,B 0,C 180,E1 -13600.264,E2 -13600.264} C_VEL
LIN {X 0,Y 354.946,Z 376.273,A -85,B 0,C 180,E1 -13604.019,E2 -13604.019} C_VEL
LIN {X 0,Y 354.926,Z 376.273,A -85,B 0,C 180,E1 -13608.109,E2 -13608.109} C_VEL
LIN {X 0,Y 354.842,Z 376.284,A -85,B 0,C 180,E1 -13612.106,E2 -13612.106} C_VEL
